LIN {X -0.105,Y -299.995,Z 1739.508,A 0.000,B 0.000,C 90.000,E1 271.547} C_DIS
LIN {X -0.094,Y -289.152,Z 1739.507,A 0.000,B 0.000,C 90.000,E1 271.260} C_DIS
LIN {X -0.103,Y -276.677,Z 1739.506,A 0.000,B 0.000,C 90.000,E1 271.031} C_DIS
LIN {X -0.110,Y -262.609,Z 1739.505,A 0.000,B 0.000,C 90.000,E1 270.859} C_DIS
LIN {X -0.020,Y -246.095,Z 1739.504,A 0.000,B 0.000,C 90.000,E1 270.688} C_DIS
LIN {X 0.079,Y -238.061,Z 1739.504,A 0.000,B 0.000,C 90.000,E1 270.630} C_DIS
LIN {X 0.025,Y -181.540,Z 1739.504,A 0.000,B 0.000,C 90.000,E1 270.630} C_DIS
LIN {X -0.061,Y -181.505,Z 1739.499,A 0.000,B 0.000,C 90.000,E1 269.771} C_DIS
LIN {X 0.044,Y -180.908,Z 1739.475,A 0.000,B 0.000,C 90.000,E1 265.527} C_DIS
LIN {X -0.079,Y -180.767,Z 1739.471,A 0.000,B 0.000,C 90.000,E1 264.723} C_DIS
LIN {X -0.008,Y -178.861,Z 1739.442,A 0.000,B 0.000,C 90.000,E1 259.634} C_DIS
LIN {X 0.064,Y -175.904,Z 1739.414,A 0.000,B 0.000,C 90.000,E1 254.519} C_DIS
LIN {X 0.003,Y -174.586,Z 1739.405,A 0.000,B 0.000,C 90.000,E1 252.834} C_DIS
LIN {X 0.037,Y -171.569,Z 1739.381,A 0.000,B 0.000,C 90.000,E1 248.539} C_DIS
LIN {X 0.019,Y -167.793,Z 1739.357,A 0.000,B 0.000,C 90.000,E1 244.229} C_DIS
LIN {X 0.033,Y -166.508,Z 1739.347,A 0.000,B 0.000,C 90.000,E1 242.487} C_DIS
LIN {X 0.029,Y -163.216,Z 1739.328,A 0.000,B 0.000,C 90.000,E1 238.997} C_DIS
LIN {X -0.006,Y -161.182,Z 1739.313,A 0.000,B 0.000,C 90.000,E1 236.373} C_DIS
LIN {X -0.006,Y -157.195,Z 1739.289,A 0.000,B 0.000,C 90.000,E1 231.949} C_DIS
LIN {X 0.040,Y -155.924,Z 1739.279,A 0.000,B 0.000,C 90.000,E1 230.150} C_DIS
LIN {X -0.011,Y -152.175,Z 1739.254,A 0.000,B 0.000,C 90.000,E1 225.688} C_DIS
LIN {X 0.005,Y -150.423,Z 1739.239,A 0.000,B 0.000,C 90.000,E1 222.975} C_DIS
LIN {X -0.070,Y -147.151,Z 1739.214,A 0.000,B 0.000,C 90.000,E1 218.463} C_DIS
LIN {X 0.018,Y -145.164,Z 1739.193,A 0.000,B 0.000,C 90.000,E1 214.771} C_DIS
LIN {X -0.066,Y -142.318,Z 1739.162,A 0.000,B 0.000,C 90.000,E1 209.283} C_DIS
LIN {X 0.054,Y -141.707,Z 1739.152,A 0.000,B 0.000,C 90.000,E1 207.385} C_DIS
LIN {X -0.023,Y -139.469,Z 1739.116,A 0.000,B 0.000,C 90.000,E1 200.918} C_DIS
LIN {X 0.031,Y -139.202,Z 1739.106,A 0.000,B 0.000,C 90.000,E1 199.033} C_DIS
LIN {X -0.042,Y -138.328,Z 1739.054,A 0.000,B 0.000,C 90.000,E1 189.726} C_DIS
LIN {X -0.039,Y -139.442,Z 1739.007,A 0.000,B 0.000,C 90.000,E1 181.318} C_DIS
LIN {X 0.040,Y -140.976,Z 1738.976,A 0.000,B 0.000,C 90.000,E1 175.698} C_DIS
LIN {X -0.010,Y -142.732,Z 1738.956,A 0.000,B 0.000,C 90.000,E1 172.008} C_DIS
LIN {X -0.053,Y -145.120,Z 1738.930,A 0.000,B 0.000,C 90.000,E1 167.409} C_DIS
LIN {X -0.058,Y -147.744,Z 1738.910,A 0.000,B 0.000,C 90.000,E1 163.740} C_DIS
LIN {X 0.023,Y -150.410,Z 1738.889,A 0.000,B 0.000,C 90.000,E1 160.061} C_DIS
LIN {X 0.038,Y -153.849,Z 1738.869,A 0.000,B 0.000,C 90.000,E1 156.433} C_DIS
LIN {X -0.044,Y -157.259,Z 1738.849,A 0.000,B 0.000,C 90.000,E1 152.871} C_DIS
LIN {X 0.034,Y -161.434,Z 1738.829,A 0.000,B 0.000,C 90.000,E1 149.282} C_DIS
LIN {X 0.041,Y -165.635,Z 1738.810,A 0.000,B 0.000,C 90.000,E1 145.754} C_DIS
LIN {X 0.024,Y -170.566,Z 1738.790,A 0.000,B 0.000,C 90.000,E1 142.271} C_DIS
LIN {X -0.069,Y -175.444,Z 1738.771,A 0.000,B 0.000,C 90.000,E1 138.852} C_DIS
LIN {X 0.047,Y -181.067,Z 1738.752,A 0.000,B 0.000,C 90.000,E1 135.405} C_DIS
LIN {X 0.038,Y -186.506,Z 1738.734,A 0.000,B 0.000,C 90.000,E1 132.043} C_DIS
LIN {X -0.020,Y -191.124,Z 1738.720,A 0.000,B 0.000,C 90.000,E1 129.564} C_DIS
LIN {X -0.099,Y -196.922,Z 1738.702,A 0.000,B 0.000,C 90.000,E1 126.297} C_DIS
LIN {X 0.095,Y -200.185,Z 1738.692,A 0.000,B 0.000,C 90.000,E1 124.612} C_DIS
LIN {X 0.091,Y -207.680,Z 1738.670,A 0.000,B 0.000,C 90.000,E1 120.590} C_DIS
LIN {X 0.056,Y -210.159,Z 1738.663,A 0.000,B 0.000,C 90.000,E1 119.411} C_DIS
LIN {X 0.030,Y -335.745,Z 1738.663,A 0.000,B 0.000,C 90.000,E1 119.411} C_DIS
LIN {X -0.088,Y -336.892,Z 1738.663,A 0.000,B 0.000,C 90.000,E1 119.411} C_DIS
LIN {X 0.032,Y -341.306,Z 1738.662,A 0.000,B 0.000,C 90.000,E1 119.205} C_DIS
LIN {X -0.012,Y -343.768,Z 1738.661,A 0.000,B 0.000,C 90.000,E1 119.027} C_DIS
LIN {X 0.124,Y -347.586,Z 1738.659,A 0.000,B 0.000,C 90.000,E1 118.565} C_DIS
LIN {X 0.008,Y -349.403,Z 1738.657,A 0.000,B 0.000,C 90.000,E1 118.281} C_DIS
LIN {X -0.092,Y -363.937,Z 1738.640,A 0.000,B 0.000,C 90.000,E1 115.283} C_DIS
LIN {X -0.172,Y -378.581,Z 1738.626,A 0.000,B 0.000,C 90.000,E1 112.642} C_DIS
LIN {X 0.064,Y -392.989,Z 1738.613,A 0.000,B 0.000,C 90.000,E1 110.301} C_DIS
LIN {X 0.021,Y -408.810,Z 1738.600,A 0.000,B 0.000,C 90.000,E1 108.055} C_DIS
LIN {X 0.119,Y -426.155,Z 1738.588,A 0.000,B 0.000,C 90.000,E1 105.843} C_DIS
LIN {X 0.012,Y -445.138,Z 1738.576,A 0.000,B 0.000,C 90.000,E1 103.716} C_DIS
LIN {X -0.048,Y -465.129,Z 1738.565,A 0.000,B 0.000,C 90.000,E1 101.715} C_DIS
LIN {X 0.245,Y -488.252,Z 1738.554,A 0.000,B 0.000,C 90.000,E1 99.613} C_DIS
LIN {X 0.198,Y -509.263,Z 1738.544,A 0.000,B 0.000,C 90.000,E1 97.936} C_DIS
LIN {X -0.014,Y -511.312,Z 1738.543,A 0.000,B 0.000,C 90.000,E1 97.757} C_DIS
LIN {X -0.101,Y -513.130,Z 1738.542,A 0.000,B 0.000,C 90.000,E1 97.530} C_DIS
LIN {X -0.123,Y -514.495,Z 1738.540,A 0.000,B 0.000,C 90.000,E1 97.296} C_DIS
LIN {X 0.246,Y -516.219,Z 1738.538,A 0.000,B 0.000,C 90.000,E1 96.777} C_DIS
LIN {X 0.109,Y -516.821,Z 1738.535,A 0.000,B 0.000,C 90.000,E1 96.315} C_DIS
LIN {X -0.018,Y -516.401,Z 1738.532,A 0.000,B 0.000,C 90.000,E1 95.853} C_DIS
LIN {X -0.144,Y -514.889,Z 1738.530,A 0.000,B 0.000,C 90.000,E1 95.391} C_DIS
LIN {X -0.231,Y -513.638,Z 1738.529,A 0.000,B 0.000,C 90.000,E1 95.163} C_DIS
LIN {X -0.048,Y -506.557,Z 1738.523,A 0.000,B 0.000,C 90.000,E1 94.188} C_DIS
LIN {X 0.214,Y -493.994,Z 1738.514,A 0.000,B 0.000,C 90.000,E1 92.465} C_DIS
LIN {X 0.190,Y -481.184,Z 1738.504,A 0.000,B 0.000,C 90.000,E1 90.745} C_DIS
LIN {X -0.083,Y -468.423,Z 1738.495,A 0.000,B 0.000,C 90.000,E1 89.026} C_DIS
LIN {X -0.131,Y -455.598,Z 1738.485,A 0.000,B 0.000,C 90.000,E1 87.249} C_DIS
LIN {X -0.184,Y -440.878,Z 1738.473,A 0.000,B 0.000,C 90.000,E1 85.179} C_DIS
LIN {X -0.140,Y -426.340,Z 1738.461,A 0.000,B 0.000,C 90.000,E1 83.053} C_DIS
LIN {X 0.132,Y -412.110,Z 1738.449,A 0.000,B 0.000,C 90.000,E1 80.849} C_DIS
LIN {X -0.002,Y -393.593,Z 1738.432,A 0.000,B 0.000,C 90.000,E1 77.813} C_DIS
LIN {X 0.145,Y -379.296,Z 1738.418,A 0.000,B 0.000,C 90.000,E1 75.227} C_DIS
LIN {X 0.106,Y -366.952,Z 1738.405,A 0.000,B 0.000,C 90.000,E1 72.906} C_DIS
LIN {X 0.045,Y -353.403,Z 1738.390,A 0.000,B 0.000,C 90.000,E1 70.242} C_DIS
LIN {X -0.120,Y -339.176,Z 1738.373,A 0.000,B 0.000,C 90.000,E1 67.230} C_DIS
LIN {X -0.058,Y -329.410,Z 1738.361,A 0.000,B 0.000,C 90.000,E1 65.049} C_DIS
LIN {X -0.200,Y -317.141,Z 1738.346,A 0.000,B 0.000,C 90.000,E1 62.231} C_DIS
LIN {X 0.050,Y -308.892,Z 1738.335,A 0.000,B 0.000,C 90.000,E1 60.255} C_DIS
LIN {X -0.098,Y -299.064,Z 1738.322,A 0.000,B 0.000,C 90.000,E1 57.995} C_DIS
LIN {X -0.130,Y -290.650,Z 1738.311,A 0.000,B 0.000,C 90.000,E1 56.008} C_DIS
LIN {X -0.073,Y -279.311,Z 1738.296,A 0.000,B 0.000,C 90.000,E1 53.290} C_DIS
LIN {X -0.108,Y -269.573,Z 1738.283,A 0.000,B 0.000,C 90.000,E1 50.884} C_DIS
LIN {X 0.030,Y -258.557,Z 1738.267,A 0.000,B 0.000,C 90.000,E1 48.038} C_DIS
LIN {X 0.032,Y -246.674,Z 1738.249,A 0.000,B 0.000,C 90.000,E1 44.798} C_DIS
LIN {X 0.070,Y -235.223,Z 1738.230,A 0.000,B 0.000,C 90.000,E1 41.472} C_DIS
LIN {X -0.002,Y -224.589,Z 1738.212,A 0.000,B 0.000,C 90.000,E1 38.096} C_DIS
LIN {X 0.061,Y -216.983,Z 1738.197,A 0.000,B 0.000,C 90.000,E1 35.391} C_DIS
LIN {X -0.014,Y -209.076,Z 1738.179,A 0.000,B 0.000,C 90.000,E1 32.291} C_DIS
LIN {X -0.045,Y -201.878,Z 1738.162,A 0.000,B 0.000,C 90.000,E1 29.127} C_DIS
LIN {X -0.026,Y -195.427,Z 1738.144,A 0.000,B 0.000,C 90.000,E1 25.899} C_DIS
LIN {X -0.061,Y -189.668,Z 1738.126,A 0.000,B 0.000,C 90.000,E1 22.642} C_DIS
LIN {X -0.030,Y -184.611,Z 1738.107,A 0.000,B 0.000,C 90.000,E1 19.322} C_DIS
LIN {X -0.010,Y -180.336,Z 1738.089,A 0.000,B 0.000,C 90.000,E1 15.969} C_DIS
LIN {X -0.016,Y -176.826,Z 1738.070,A 0.000,B 0.000,C 90.000,E1 12.591} C_DIS
LIN {X -0.049,Y -173.545,Z 1738.046,A 0.000,B 0.000,C 90.000,E1 8.341} C_DIS
LIN {X 0.048,Y -170.771,Z 1738.018,A 0.000,B 0.000,C 90.000,E1 3.154} C_DIS
LIN {X 0.062,Y -169.444,Z 1737.973,A 0.000,B 0.000,C 90.000,E1 355.184} C_DIS
LIN {X 0.057,Y -170.840,Z 1737.925,A 0.000,B 0.000,C 90.000,E1 346.533} C_DIS
LIN {X -0.063,Y -173.212,Z 1737.897,A 0.000,B 0.000,C 90.000,E1 341.402} C_DIS
LIN {X -0.019,Y -176.360,Z 1737.873,A 0.000,B 0.000,C 90.000,E1 337.102} C_DIS
LIN {X -0.085,Y -180.284,Z 1737.849,A 0.000,B 0.000,C 90.000,E1 332.871} C_DIS
LIN {X 0.040,Y -184.267,Z 1737.830,A 0.000,B 0.000,C 90.000,E1 329.459} C_DIS
LIN {X -0.017,Y -189.155,Z 1737.812,A 0.000,B 0.000,C 90.000,E1 326.135} C_DIS
LIN {X -0.060,Y -194.994,Z 1737.793,A 0.000,B 0.000,C 90.000,E1 322.844} C_DIS
LIN {X 0.072,Y -200.201,Z 1737.780,A 0.000,B 0.000,C 90.000,E1 320.356} C_DIS
LIN {X 0.032,Y -208.197,Z 1737.762,A 0.000,B 0.000,C 90.000,E1 317.148} C_DIS
LIN {X -0.005,Y -216.267,Z 1737.747,A 0.000,B 0.000,C 90.000,E1 314.393} C_DIS
LIN {X -0.010,Y -222.842,Z 1737.736,A 0.000,B 0.000,C 90.000,E1 312.447} C_DIS
LIN {X -0.110,Y -231.851,Z 1737.723,A 0.000,B 0.000,C 90.000,E1 310.172} C_DIS
LIN {X 0.024,Y -240.419,Z 1737.713,A 0.000,B 0.000,C 90.000,E1 308.257} C_DIS
LIN {X 0.160,Y -251.924,Z 1737.700,A 0.000,B 0.000,C 90.000,E1 306.011} C_DIS
LIN {X 0.122,Y -266.927,Z 1737.686,A 0.000,B 0.000,C 90.000,E1 303.499} C_DIS
LIN {X 0.083,Y -285.648,Z 1737.671,A 0.000,B 0.000,C 90.000,E1 300.718} C_DIS
LIN {X 0.081,Y -303.306,Z 1737.658,A 0.000,B 0.000,C 90.000,E1 298.359} C_DIS
LIN {X -0.094,Y -321.696,Z 1737.645,A 0.000,B 0.000,C 90.000,E1 296.104} C_DIS
LIN {X -0.079,Y -334.482,Z 1737.636,A 0.000,B 0.000,C 90.000,E1 294.567} C_DIS
LIN {X -0.023,Y -347.643,Z 1737.628,A 0.000,B 0.000,C 90.000,E1 293.003} C_DIS
LIN {X 0.095,Y -357.760,Z 1737.621,A 0.000,B 0.000,C 90.000,E1 291.770} C_DIS
LIN {X -0.150,Y -367.553,Z 1737.614,A 0.000,B 0.000,C 90.000,E1 290.610} C_DIS
LIN {X -0.022,Y -374.523,Z 1737.609,A 0.000,B 0.000,C 90.000,E1 289.704} C_DIS
LIN {X 0.183,Y -378.791,Z 1737.606,A 0.000,B 0.000,C 90.000,E1 289.087} C_DIS
LIN {X -0.066,Y -382.655,Z 1737.603,A 0.000,B 0.000,C 90.000,E1 288.544} C_DIS
LIN {X 0.071,Y -386.084,Z 1737.600,A 0.000,B 0.000,C 90.000,E1 287.946} C_DIS
LIN {X -0.136,Y -389.068,Z 1737.597,A 0.000,B 0.000,C 90.000,E1 287.402} C_DIS
LIN {X 0.047,Y -391.609,Z 1737.593,A 0.000,B 0.000,C 90.000,E1 286.804} C_DIS
LIN {X -0.078,Y -394.658,Z 1737.589,A 0.000,B 0.000,C 90.000,E1 285.969} C_DIS
LIN {X 0.139,Y -396.227,Z 1737.585,A 0.000,B 0.000,C 90.000,E1 285.371} C_DIS
LIN {X -0.017,Y -397.450,Z 1737.582,A 0.000,B 0.000,C 90.000,E1 284.828} C_DIS
LIN {X 0.118,Y -398.340,Z 1737.579,A 0.000,B 0.000,C 90.000,E1 284.245} C_DIS
LIN {X -0.027,Y -398.898,Z 1737.576,A 0.000,B 0.000,C 90.000,E1 283.703} C_DIS
LIN {X 0.125,Y -399.041,Z 1737.573,A 0.000,B 0.000,C 90.000,E1 283.119} C_DIS
LIN {X -0.107,Y -398.829,Z 1737.570,A 0.000,B 0.000,C 90.000,E1 282.591} C_DIS
LIN {X 0.052,Y -398.155,Z 1737.567,A 0.000,B 0.000,C 90.000,E1 282.007} C_DIS
LIN {X -0.178,Y -397.045,Z 1737.564,A 0.000,B 0.000,C 90.000,E1 281.478} C_DIS
LIN {X -0.025,Y -395.355,Z 1737.561,A 0.000,B 0.000,C 90.000,E1 280.894} C_DIS
LIN {X 0.120,Y -393.108,Z 1737.557,A 0.000,B 0.000,C 90.000,E1 280.310} C_DIS
LIN {X -0.139,Y -390.215,Z 1737.554,A 0.000,B 0.000,C 90.000,E1 279.782} C_DIS
LIN {X -0.026,Y -381.971,Z 1737.546,A 0.000,B 0.000,C 90.000,E1 278.341} C_DIS
LIN {X 0.051,Y -377.336,Z 1737.542,A 0.000,B 0.000,C 90.000,E1 277.466} C_DIS
LIN {X 0.027,Y -373.748,Z 1737.538,A 0.000,B 0.000,C 90.000,E1 276.891} C_DIS
LIN {X -0.017,Y -369.584,Z 1737.535,A 0.000,B 0.000,C 90.000,E1 276.315} C_DIS
LIN {X -0.080,Y -364.671,Z 1737.532,A 0.000,B 0.000,C 90.000,E1 275.739} C_DIS
LIN {X -0.168,Y -358.972,Z 1737.529,A 0.000,B 0.000,C 90.000,E1 275.163} C_DIS
LIN {X 0.052,Y -353.211,Z 1737.526,A 0.000,B 0.000,C 90.000,E1 274.588} C_DIS
LIN {X 0.112,Y -344.344,Z 1737.521,A 0.000,B 0.000,C 90.000,E1 273.841} C_DIS
LIN {X 0.146,Y -338.207,Z 1737.519,A 0.000,B 0.000,C 90.000,E1 273.383} C_DIS
LIN {X 0.047,Y -331.920,Z 1737.517,A 0.000,B 0.000,C 90.000,E1 272.980} C_DIS
LIN {X 0.117,Y -325.356,Z 1737.514,A 0.000,B 0.000,C 90.000,E1 272.579} C_DIS
LIN {X 0.077,Y -318.598,Z 1737.512,A 0.000,B 0.000,C 90.000,E1 272.236} C_DIS
LIN {X -0.028,Y -311.635,Z 1737.511,A 0.000,B 0.000,C 90.000,E1 271.949} C_DIS
LIN {X 0.119,Y -304.471,Z 1737.509,A 0.000,B 0.000,C 90.000,E1 271.661} C_DIS
LIN {X -0.056,Y -293.557,Z 1737.508,A 0.000,B 0.000,C 90.000,E1 271.375} C_DIS
LIN {X -0.060,Y -286.006,Z 1737.507,A 0.000,B 0.000,C 90.000,E1 271.203} C_DIS
LIN {X 0.065,Y -273.757,Z 1737.505,A 0.000,B 0.000,C 90.000,E1 270.974} C_DIS
LIN {X 0.066,Y -259.464,Z 1737.505,A 0.000,B 0.000,C 90.000,E1 270.802} C_DIS
LIN {X 0.016,Y -243.753,Z 1737.504,A 0.000,B 0.000,C 90.000,E1 270.688} C_DIS
LIN {X -0.077,Y -236.046,Z 1737.504,A 0.000,B 0.000,C 90.000,E1 270.688} C_DIS
LIN {X 0.087,Y -181.536,Z 1737.504,A 0.000,B 0.000,C 90.000,E1 270.630} C_DIS
LIN {X 0.037,Y -181.513,Z 1737.499,A 0.000,B 0.000,C 90.000,E1 269.771} C_DIS
LIN {X -0.039,Y -180.908,Z 1737.475,A 0.000,B 0.000,C 90.000,E1 265.584} C_DIS
LIN {X 0.019,Y -180.779,Z 1737.471,A 0.000,B 0.000,C 90.000,E1 264.723} C_DIS
LIN {X -0.087,Y -178.875,Z 1737.443,A 0.000,B 0.000,C 90.000,E1 259.690} C_DIS
LIN {X -0.010,Y -175.918,Z 1737.414,A 0.000,B 0.000,C 90.000,E1 254.574} C_DIS
LIN {X 0.046,Y -174.613,Z 1737.405,A 0.000,B 0.000,C 90.000,E1 252.851} C_DIS
LIN {X -0.028,Y -171.593,Z 1737.381,A 0.000,B 0.000,C 90.000,E1 248.592} C_DIS
LIN {X -0.039,Y -167.815,Z 1737.357,A 0.000,B 0.000,C 90.000,E1 244.280} C_DIS
LIN {X -0.021,Y -166.538,Z 1737.347,A 0.000,B 0.000,C 90.000,E1 242.538} C_DIS
LIN {X 0.028,Y -162.536,Z 1737.323,A 0.000,B 0.000,C 90.000,E1 238.152} C_DIS
LIN {X -0.050,Y -161.212,Z 1737.313,A 0.000,B 0.000,C 90.000,E1 236.421} C_DIS
LIN {X -0.014,Y -157.220,Z 1737.289,A 0.000,B 0.000,C 90.000,E1 231.984} C_DIS
LIN {X 0.009,Y -155.946,Z 1737.279,A 0.000,B 0.000,C 90.000,E1 230.194} C_DIS
LIN {X -0.032,Y -152.199,Z 1737.254,A 0.000,B 0.000,C 90.000,E1 225.729} C_DIS
LIN {X -0.010,Y -150.444,Z 1737.239,A 0.000,B 0.000,C 90.000,E1 223.014} C_DIS
LIN {X 0.016,Y -147.171,Z 1737.214,A 0.000,B 0.000,C 90.000,E1 218.463} C_DIS
LIN {X -0.016,Y -145.187,Z 1737.193,A 0.000,B 0.000,C 90.000,E1 214.818} C_DIS
LIN {X 0.018,Y -142.331,Z 1737.163,A 0.000,B 0.000,C 90.000,E1 209.283} C_DIS
LIN {X -0.053,Y -141.719,Z 1737.152,A 0.000,B 0.000,C 90.000,E1 207.462} C_DIS
LIN {X 0.060,Y -139.476,Z 1737.116,A 0.000,B 0.000,C 90.000,E1 200.918} C_DIS
LIN {X 0.051,Y -138.973,Z 1737.101,A 0.000,B 0.000,C 90.000,E1 198.127} C_DIS
LIN {X 0.040,Y -138.331,Z 1737.054,A 0.000,B 0.000,C 90.000,E1 189.726} C_DIS
LIN {X 0.044,Y -139.434,Z 1737.007,A 0.000,B 0.000,C 90.000,E1 181.318} C_DIS
LIN {X -0.016,Y -140.963,Z 1736.976,A 0.000,B 0.000,C 90.000,E1 175.755} C_DIS
LIN {X 0.074,Y -142.719,Z 1736.956,A 0.000,B 0.000,C 90.000,E1 172.008} C_DIS
LIN {X 0.033,Y -145.098,Z 1736.930,A 0.000,B 0.000,C 90.000,E1 167.409} C_DIS
LIN {X 0.029,Y -147.723,Z 1736.910,A 0.000,B 0.000,C 90.000,E1 163.740} C_DIS
LIN {X -0.032,Y -150.382,Z 1736.889,A 0.000,B 0.000,C 90.000,E1 160.115} C_DIS
LIN {X -0.013,Y -153.813,Z 1736.869,A 0.000,B 0.000,C 90.000,E1 156.485} C_DIS
LIN {X 0.046,Y -157.224,Z 1736.849,A 0.000,B 0.000,C 90.000,E1 152.871} C_DIS
LIN {X -0.014,Y -161.392,Z 1736.830,A 0.000,B 0.000,C 90.000,E1 149.331} C_DIS
LIN {X -0.003,Y -165.594,Z 1736.810,A 0.000,B 0.000,C 90.000,E1 145.801} C_DIS
LIN {X -0.017,Y -170.517,Z 1736.791,A 0.000,B 0.000,C 90.000,E1 142.316} C_DIS
LIN {X 0.027,Y -175.396,Z 1736.771,A 0.000,B 0.000,C 90.000,E1 138.852} C_DIS
LIN {X 0.018,Y -181.021,Z 1736.753,A 0.000,B 0.000,C 90.000,E1 135.445} C_DIS
LIN {X 0.012,Y -186.452,Z 1736.734,A 0.000,B 0.000,C 90.000,E1 132.081} C_DIS
LIN {X 0.081,Y -191.076,Z 1736.720,A 0.000,B 0.000,C 90.000,E1 129.564} C_DIS
LIN {X 0.004,Y -196.865,Z 1736.702,A 0.000,B 0.000,C 90.000,E1 126.297} C_DIS
LIN {X -0.080,Y -200.123,Z 1736.693,A 0.000,B 0.000,C 90.000,E1 124.692} C_DIS
LIN {X -0.087,Y -207.620,Z 1736.670,A 0.000,B 0.000,C 90.000,E1 120.669} C_DIS
LIN {X -0.021,Y -210.103,Z 1736.664,A 0.000,B 0.000,C 90.000,E1 119.461} C_DIS
LIN {X -0.093,Y -335.517,Z 1736.664,A 0.000,B 0.000,C 90.000,E1 119.461} C_DIS
LIN {X 0.081,Y -336.703,Z 1736.663,A 0.000,B 0.000,C 90.000,E1 119.411} C_DIS
LIN {X 0.205,Y -341.146,Z 1736.662,A 0.000,B 0.000,C 90.000,E1 119.205} C_DIS
LIN {X -0.139,Y -343.611,Z 1736.661,A 0.000,B 0.000,C 90.000,E1 119.077} C_DIS
LIN {X -0.001,Y -347.427,Z 1736.659,A 0.000,B 0.000,C 90.000,E1 118.615} C_DIS
LIN {X 0.024,Y -349.245,Z 1736.657,A 0.000,B 0.000,C 90.000,E1 118.309} C_DIS
LIN {X 0.093,Y -363.763,Z 1736.641,A 0.000,B 0.000,C 90.000,E1 115.283} C_DIS
LIN {X 0.015,Y -378.390,Z 1736.626,A 0.000,B 0.000,C 90.000,E1 112.642} C_DIS
LIN {X -0.114,Y -392.781,Z 1736.613,A 0.000,B 0.000,C 90.000,E1 110.355} C_DIS
LIN {X 0.213,Y -408.585,Z 1736.600,A 0.000,B 0.000,C 90.000,E1 108.055} C_DIS
LIN {X -0.096,Y -425.910,Z 1736.588,A 0.000,B 0.000,C 90.000,E1 105.898} C_DIS
LIN {X -0.226,Y -444.875,Z 1736.576,A 0.000,B 0.000,C 90.000,E1 103.772} C_DIS
LIN {X 0.138,Y -464.859,Z 1736.565,A 0.000,B 0.000,C 90.000,E1 101.715} C_DIS
LIN {X -0.060,Y -487.976,Z 1736.554,A 0.000,B 0.000,C 90.000,E1 99.670} C_DIS
LIN {X -0.137,Y -508.985,Z 1736.544,A 0.000,B 0.000,C 90.000,E1 97.992} C_DIS
LIN {X 0.154,Y -511.042,Z 1736.543,A 0.000,B 0.000,C 90.000,E1 97.757} C_DIS
LIN {X 0.069,Y -512.860,Z 1736.542,A 0.000,B 0.000,C 90.000,E1 97.530} C_DIS
LIN {X 0.052,Y -514.227,Z 1736.541,A 0.000,B 0.000,C 90.000,E1 97.296} C_DIS
LIN {X -0.093,Y -515.957,Z 1736.538,A 0.000,B 0.000,C 90.000,E1 96.834} C_DIS
LIN {X -0.231,Y -516.566,Z 1736.535,A 0.000,B 0.000,C 90.000,E1 96.372} C_DIS
LIN {X 0.152,Y -516.154,Z 1736.533,A 0.000,B 0.000,C 90.000,E1 95.853} C_DIS
LIN {X 0.025,Y -514.651,Z 1736.530,A 0.000,B 0.000,C 90.000,E1 95.391} C_DIS
LIN {X -0.063,Y -513.406,Z 1736.529,A 0.000,B 0.000,C 90.000,E1 95.163} C_DIS
LIN {X 0.114,Y -506.330,Z 1736.523,A 0.000,B 0.000,C 90.000,E1 94.188} C_DIS
LIN {X -0.126,Y -493.770,Z 1736.514,A 0.000,B 0.000,C 90.000,E1 92.522} C_DIS
LIN {X -0.145,Y -480.954,Z 1736.504,A 0.000,B 0.000,C 90.000,E1 90.802} C_DIS
LIN {X 0.055,Y -468.194,Z 1736.495,A 0.000,B 0.000,C 90.000,E1 89.026} C_DIS
LIN {X -0.001,Y -455.379,Z 1736.485,A 0.000,B 0.000,C 90.000,E1 87.249} C_DIS
LIN {X 0.162,Y -442.465,Z 1736.475,A 0.000,B 0.000,C 90.000,E1 85.412} C_DIS
LIN {X 0.092,Y -429.699,Z 1736.464,A 0.000,B 0.000,C 90.000,E1 83.571} C_DIS
LIN {X -0.177,Y -417.136,Z 1736.454,A 0.000,B 0.000,C 90.000,E1 81.724} C_DIS
LIN {X 0.155,Y -398.215,Z 1736.437,A 0.000,B 0.000,C 90.000,E1 78.645} C_DIS
LIN {X 0.039,Y -383.704,Z 1736.423,A 0.000,B 0.000,C 90.000,E1 76.117} C_DIS
LIN {X 0.108,Y -371.237,Z 1736.410,A 0.000,B 0.000,C 90.000,E1 73.795} C_DIS
LIN {X -0.011,Y -359.030,Z 1736.397,A 0.000,B 0.000,C 90.000,E1 71.456} C_DIS
LIN {X -0.132,Y -344.398,Z 1736.380,A 0.000,B 0.000,C 90.000,E1 68.465} C_DIS
LIN {X -0.086,Y -334.637,Z 1736.368,A 0.000,B 0.000,C 90.000,E1 66.305} C_DIS
LIN {X 0.060,Y -322.128,Z 1736.353,A 0.000,B 0.000,C 90.000,E1 63.461} C_DIS
LIN {X -0.030,Y -313.999,Z 1736.342,A 0.000,B 0.000,C 90.000,E1 61.563} C_DIS
LIN {X 0.045,Y -304.268,Z 1736.329,A 0.000,B 0.000,C 90.000,E1 59.282} C_DIS
LIN {X -0.048,Y -294.502,Z 1736.317,A 0.000,B 0.000,C 90.000,E1 56.993} C_DIS
LIN {X -0.009,Y -286.033,Z 1736.305,A 0.000,B 0.000,C 90.000,E1 54.975} C_DIS
LIN {X -0.130,Y -274.840,Z 1736.290,A 0.000,B 0.000,C 90.000,E1 52.271} C_DIS
LIN {X -0.094,Y -265.096,Z 1736.277,A 0.000,B 0.000,C 90.000,E1 49.828} C_DIS
LIN {X -0.084,Y -254.181,Z 1736.261,A 0.000,B 0.000,C 90.000,E1 46.986} C_DIS
LIN {X 0.166,Y -243.715,Z 1736.245,A 0.000,B 0.000,C 90.000,E1 44.028} C_DIS
LIN {X -0.054,Y -232.449,Z 1736.226,A 0.000,B 0.000,C 90.000,E1 40.744} C_DIS
LIN {X 0.006,Y -222.009,Z 1736.207,A 0.000,B 0.000,C 90.000,E1 37.317} C_DIS
LIN {X 0.022,Y -214.644,Z 1736.192,A 0.000,B 0.000,C 90.000,E1 34.612} C_DIS
LIN {X 0.062,Y -206.948,Z 1736.175,A 0.000,B 0.000,C 90.000,E1 31.465} C_DIS
LIN {X 0.047,Y -199.982,Z 1736.157,A 0.000,B 0.000,C 90.000,E1 28.281} C_DIS
LIN {X -0.068,Y -193.740,Z 1736.139,A 0.000,B 0.000,C 90.000,E1 25.079} C_DIS
LIN {X 0.030,Y -188.141,Z 1736.121,A 0.000,B 0.000,C 90.000,E1 21.770} C_DIS
LIN {X -0.045,Y -183.331,Z 1736.103,A 0.000,B 0.000,C 90.000,E1 18.471} C_DIS
LIN {X -0.108,Y -179.237,Z 1736.084,A 0.000,B 0.000,C 90.000,E1 15.134} C_DIS
LIN {X -0.008,Y -175.952,Z 1736.065,A 0.000,B 0.000,C 90.000,E1 11.715} C_DIS
LIN {X -0.072,Y -172.842,Z 1736.041,A 0.000,B 0.000,C 90.000,E1 7.466} C_DIS
LIN {X -0.038,Y -170.324,Z 1736.013,A 0.000,B 0.000,C 90.000,E1 2.293} C_DIS
LIN {X 0.057,Y -169.274,Z 1735.969,A 0.000,B 0.000,C 90.000,E1 354.318} C_DIS
LIN {X -0.049,Y -170.993,Z 1735.920,A 0.000,B 0.000,C 90.000,E1 345.700} C_DIS
LIN {X 0.055,Y -173.609,Z 1735.892,A 0.000,B 0.000,C 90.000,E1 340.496} C_DIS
LIN {X 0.015,Y -176.980,Z 1735.868,A 0.000,B 0.000,C 90.000,E1 336.230} C_DIS
LIN {X 0.045,Y -181.115,Z 1735.844,A 0.000,B 0.000,C 90.000,E1 331.975} C_DIS
LIN {X 0.029,Y -185.352,Z 1735.826,A 0.000,B 0.000,C 90.000,E1 328.614} C_DIS
LIN {X -0.061,Y -190.485,Z 1735.807,A 0.000,B 0.000,C 90.000,E1 325.308} C_DIS
LIN {X -0.095,Y -195.037,Z 1735.793,A 0.000,B 0.000,C 90.000,E1 322.844} C_DIS
LIN {X 0.052,Y -202.180,Z 1735.775,A 0.000,B 0.000,C 90.000,E1 319.542} C_DIS
LIN {X 0.032,Y -209.428,Z 1735.760,A 0.000,B 0.000,C 90.000,E1 316.743} C_DIS
LIN {X 0.124,Y -216.432,Z 1735.747,A 0.000,B 0.000,C 90.000,E1 314.352} C_DIS
LIN {X -0.034,Y -223.033,Z 1735.736,A 0.000,B 0.000,C 90.000,E1 312.447} C_DIS
LIN {X -0.074,Y -230.467,Z 1735.725,A 0.000,B 0.000,C 90.000,E1 310.539} C_DIS
LIN {X 0.032,Y -238.788,Z 1735.715,A 0.000,B 0.000,C 90.000,E1 308.624} C_DIS
LIN {X -0.066,Y -250.065,Z 1735.702,A 0.000,B 0.000,C 90.000,E1 306.423} C_DIS
LIN {X -0.079,Y -260.471,Z 1735.692,A 0.000,B 0.000,C 90.000,E1 304.612} C_DIS
LIN {X 0.088,Y -278.636,Z 1735.677,A 0.000,B 0.000,C 90.000,E1 301.750} C_DIS
LIN {X 0.068,Y -298.424,Z 1735.661,A 0.000,B 0.000,C 90.000,E1 299.027} C_DIS
LIN {X -0.009,Y -319.260,Z 1735.647,A 0.000,B 0.000,C 90.000,E1 296.411} C_DIS
LIN {X -0.149,Y -331.997,Z 1735.638,A 0.000,B 0.000,C 90.000,E1 294.899} C_DIS
LIN {X -0.110,Y -345.202,Z 1735.630,A 0.000,B 0.000,C 90.000,E1 293.334} C_DIS
LIN {X 0.090,Y -355.417,Z 1735.623,A 0.000,B 0.000,C 90.000,E1 292.078} C_DIS
LIN {X -0.121,Y -367.725,Z 1735.614,A 0.000,B 0.000,C 90.000,E1 290.610} C_DIS
LIN {X 0.009,Y -374.708,Z 1735.609,A 0.000,B 0.000,C 90.000,E1 289.704} C_DIS
LIN {X -0.141,Y -378.989,Z 1735.606,A 0.000,B 0.000,C 90.000,E1 289.141} C_DIS
LIN {X 0.091,Y -384.629,Z 1735.601,A 0.000,B 0.000,C 90.000,E1 288.236} C_DIS
LIN {X -0.126,Y -387.809,Z 1735.598,A 0.000,B 0.000,C 90.000,E1 287.692} C_DIS
LIN {X 0.046,Y -390.589,Z 1735.595,A 0.000,B 0.000,C 90.000,E1 287.094} C_DIS
LIN {X -0.137,Y -392.943,Z 1735.592,A 0.000,B 0.000,C 90.000,E1 286.551} C_DIS
LIN {X -0.038,Y -394.879,Z 1735.589,A 0.000,B 0.000,C 90.000,E1 285.969} C_DIS
LIN {X -0.201,Y -396.449,Z 1735.586,A 0.000,B 0.000,C 90.000,E1 285.426} C_DIS
LIN {X 0.026,Y -397.685,Z 1735.582,A 0.000,B 0.000,C 90.000,E1 284.828} C_DIS
LIN {X 0.164,Y -398.578,Z 1735.579,A 0.000,B 0.000,C 90.000,E1 284.245} C_DIS
LIN {X 0.020,Y -399.122,Z 1735.576,A 0.000,B 0.000,C 90.000,E1 283.703} C_DIS
LIN {X 0.173,Y -399.270,Z 1735.573,A 0.000,B 0.000,C 90.000,E1 283.119} C_DIS
LIN {X -0.057,Y -399.089,Z 1735.570,A 0.000,B 0.000,C 90.000,E1 282.591} C_DIS
LIN {X 0.103,Y -398.421,Z 1735.567,A 0.000,B 0.000,C 90.000,E1 282.007} C_DIS
LIN {X -0.127,Y -397.299,Z 1735.564,A 0.000,B 0.000,C 90.000,E1 281.478} C_DIS
LIN {X 0.028,Y -395.595,Z 1735.561,A 0.000,B 0.000,C 90.000,E1 280.894} C_DIS
LIN {X 0.175,Y -393.392,Z 1735.557,A 0.000,B 0.000,C 90.000,E1 280.310} C_DIS
LIN {X -0.149,Y -390.578,Z 1735.554,A 0.000,B 0.000,C 90.000,E1 279.792} C_DIS
LIN {X 0.055,Y -382.308,Z 1735.546,A 0.000,B 0.000,C 90.000,E1 278.341} C_DIS
LIN {X 0.108,Y -377.600,Z 1735.542,A 0.000,B 0.000,C 90.000,E1 277.473} C_DIS
LIN {X 0.132,Y -373.983,Z 1735.538,A 0.000,B 0.000,C 90.000,E1 276.891} C_DIS
LIN {X 0.090,Y -369.788,Z 1735.535,A 0.000,B 0.000,C 90.000,E1 276.315} C_DIS
LIN {X 0.026,Y -364.885,Z 1735.532,A 0.000,B 0.000,C 90.000,E1 275.739} C_DIS
LIN {X -0.063,Y -359.207,Z 1735.529,A 0.000,B 0.000,C 90.000,E1 275.163} C_DIS
LIN {X 0.002,Y -350.518,Z 1735.524,A 0.000,B 0.000,C 90.000,E1 274.359} C_DIS
LIN {X -0.070,Y -344.678,Z 1735.522,A 0.000,B 0.000,C 90.000,E1 273.898} C_DIS
LIN {X 0.130,Y -335.598,Z 1735.518,A 0.000,B 0.000,C 90.000,E1 273.212} C_DIS
LIN {X 0.090,Y -329.117,Z 1735.516,A 0.000,B 0.000,C 90.000,E1 272.808} C_DIS
LIN {X -0.064,Y -322.435,Z 1735.514,A 0.000,B 0.000,C 90.000,E1 272.465} C_DIS
LIN {X 0.013,Y -315.507,Z 1735.512,A 0.000,B 0.000,C 90.000,E1 272.121} C_DIS
LIN {X 0.033,Y -308.539,Z 1735.510,A 0.000,B 0.000,C 90.000,E1 271.835} C_DIS
LIN {X 0.033,Y -297.863,Z 1735.508,A 0.000,B 0.000,C 90.000,E1 271.489} C_DIS
LIN {X -0.054,Y -290.662,Z 1735.507,A 0.000,B 0.000,C 90.000,E1 271.318} C_DIS
LIN {X -0.051,Y -278.551,Z 1735.506,A 0.000,B 0.000,C 90.000,E1 271.088} C_DIS
LIN {X -0.088,Y -265.066,Z 1735.505,A 0.000,B 0.000,C 90.000,E1 270.917} C_DIS
LIN {X -0.045,Y -255.020,Z 1735.504,A 0.000,B 0.000,C 90.000,E1 270.802} C_DIS
LIN {X 0.046,Y -239.872,Z 1735.504,A 0.000,B 0.000,C 90.000,E1 270.688} C_DIS
LIN {X 0.001,Y -181.529,Z 1735.504,A 0.000,B 0.000,C 90.000,E1 270.688} C_DIS
LIN {X -0.046,Y -181.522,Z 1735.499,A 0.000,B 0.000,C 90.000,E1 269.828} C_DIS
LIN {X -0.063,Y -180.791,Z 1735.471,A 0.000,B 0.000,C 90.000,E1 264.780} C_DIS
LIN {X 0.011,Y -178.888,Z 1735.443,A 0.000,B 0.000,C 90.000,E1 259.690} C_DIS
LIN {X 0.087,Y -175.932,Z 1735.414,A 0.000,B 0.000,C 90.000,E1 254.574} C_DIS
LIN {X 0.033,Y -175.377,Z 1735.410,A 0.000,B 0.000,C 90.000,E1 253.740} C_DIS
LIN {X 0.030,Y -172.151,Z 1735.386,A 0.000,B 0.000,C 90.000,E1 249.464} C_DIS
LIN {X 0.067,Y -171.617,Z 1735.381,A 0.000,B 0.000,C 90.000,E1 248.592} C_DIS
LIN {X 0.055,Y -167.840,Z 1735.357,A 0.000,B 0.000,C 90.000,E1 244.280} C_DIS
LIN {X -0.004,Y -166.568,Z 1735.348,A 0.000,B 0.000,C 90.000,E1 242.564} C_DIS
LIN {X -0.018,Y -162.561,Z 1735.323,A 0.000,B 0.000,C 90.000,E1 238.201} C_DIS
LIN {X 0.042,Y -161.241,Z 1735.313,A 0.000,B 0.000,C 90.000,E1 236.421} C_DIS
LIN {X -0.047,Y -157.245,Z 1735.289,A 0.000,B 0.000,C 90.000,E1 232.029} C_DIS
LIN {X -0.001,Y -155.968,Z 1735.279,A 0.000,B 0.000,C 90.000,E1 230.231} C_DIS
LIN {X 0.057,Y -152.223,Z 1735.254,A 0.000,B 0.000,C 90.000,E1 225.729} C_DIS
LIN {X -0.032,Y -150.466,Z 1735.239,A 0.000,B 0.000,C 90.000,E1 223.056} C_DIS
LIN {X -0.012,Y -147.191,Z 1735.214,A 0.000,B 0.000,C 90.000,E1 218.508} C_DIS
LIN {X 0.069,Y -145.210,Z 1735.194,A 0.000,B 0.000,C 90.000,E1 214.818} C_DIS
LIN {X -0.021,Y -142.343,Z 1735.163,A 0.000,B 0.000,C 90.000,E1 209.333} C_DIS
LIN {X 0.032,Y -141.731,Z 1735.153,A 0.000,B 0.000,C 90.000,E1 207.462} C_DIS
LIN {X 0.014,Y -139.483,Z 1735.117,A 0.000,B 0.000,C 90.000,E1 200.972} C_DIS
LIN {X 0.003,Y -138.983,Z 1735.101,A 0.000,B 0.000,C 90.000,E1 198.181} C_DIS
LIN {X -0.035,Y -138.333,Z 1735.054,A 0.000,B 0.000,C 90.000,E1 189.792} C_DIS
LIN {X -0.012,Y -139.426,Z 1735.008,A 0.000,B 0.000,C 90.000,E1 181.375} C_DIS
LIN {X 0.042,Y -141.351,Z 1734.971,A 0.000,B 0.000,C 90.000,E1 174.837} C_DIS
LIN {X 0.019,Y -142.705,Z 1734.956,A 0.000,B 0.000,C 90.000,E1 172.064} C_DIS
LIN {X -0.023,Y -145.077,Z 1734.930,A 0.000,B 0.000,C 90.000,E1 167.465} C_DIS
LIN {X -0.027,Y -147.702,Z 1734.910,A 0.000,B 0.000,C 90.000,E1 163.795} C_DIS
LIN {X 0.006,Y -150.354,Z 1734.890,A 0.000,B 0.000,C 90.000,E1 160.134} C_DIS
LIN {X 0.076,Y -153.778,Z 1734.870,A 0.000,B 0.000,C 90.000,E1 156.485} C_DIS
LIN {X -0.003,Y -157.190,Z 1734.850,A 0.000,B 0.000,C 90.000,E1 152.922} C_DIS
LIN {X 0.078,Y -161.349,Z 1734.830,A 0.000,B 0.000,C 90.000,E1 149.331} C_DIS
LIN {X 0.090,Y -165.552,Z 1734.810,A 0.000,B 0.000,C 90.000,E1 145.801} C_DIS
LIN {X -0.025,Y -170.467,Z 1734.791,A 0.000,B 0.000,C 90.000,E1 142.351} C_DIS
LIN {X -0.008,Y -175.348,Z 1734.772,A 0.000,B 0.000,C 90.000,E1 138.895} C_DIS
LIN {X -0.012,Y -180.973,Z 1734.753,A 0.000,B 0.000,C 90.000,E1 135.486} C_DIS
LIN {X -0.024,Y -186.397,Z 1734.734,A 0.000,B 0.000,C 90.000,E1 132.123} C_DIS
LIN {X -0.085,Y -191.025,Z 1734.720,A 0.000,B 0.000,C 90.000,E1 129.644} C_DIS
LIN {X 0.107,Y -196.807,Z 1734.702,A 0.000,B 0.000,C 90.000,E1 126.297} C_DIS
LIN {X 0.026,Y -200.060,Z 1734.693,A 0.000,B 0.000,C 90.000,E1 124.692} C_DIS
LIN {X 0.020,Y -207.560,Z 1734.670,A 0.000,B 0.000,C 90.000,E1 120.669} C_DIS
LIN {X -0.017,Y -210.045,Z 1734.664,A 0.000,B 0.000,C 90.000,E1 119.489} C_DIS
LIN {X 0.078,Y -335.262,Z 1734.664,A 0.000,B 0.000,C 90.000,E1 119.461} C_DIS
LIN {X -0.040,Y -336.493,Z 1734.664,A 0.000,B 0.000,C 90.000,E1 119.461} C_DIS
LIN {X -0.085,Y -340.971,Z 1734.663,A 0.000,B 0.000,C 90.000,E1 119.283} C_DIS
LIN {X 0.038,Y -343.444,Z 1734.662,A 0.000,B 0.000,C 90.000,E1 119.077} C_DIS
LIN {X 0.186,Y -347.259,Z 1734.659,A 0.000,B 0.000,C 90.000,E1 118.615} C_DIS
LIN {X -0.093,Y -349.079,Z 1734.657,A 0.000,B 0.000,C 90.000,E1 118.359} C_DIS
LIN {X 0.023,Y -365.127,Z 1734.639,A 0.000,B 0.000,C 90.000,E1 115.027} C_DIS
LIN {X -0.017,Y -379.909,Z 1734.624,A 0.000,B 0.000,C 90.000,E1 112.386} C_DIS
LIN {X 0.117,Y -394.452,Z 1734.612,A 0.000,B 0.000,C 90.000,E1 110.066} C_DIS
LIN {X 0.119,Y -410.420,Z 1734.599,A 0.000,B 0.000,C 90.000,E1 107.819} C_DIS
LIN {X -0.146,Y -427.922,Z 1734.587,A 0.000,B 0.000,C 90.000,E1 105.662} C_DIS
LIN {X -0.199,Y -447.045,Z 1734.575,A 0.000,B 0.000,C 90.000,E1 103.536} C_DIS
LIN {X -0.139,Y -467.094,Z 1734.564,A 0.000,B 0.000,C 90.000,E1 101.535} C_DIS
LIN {X 0.187,Y -490.299,Z 1734.553,A 0.000,B 0.000,C 90.000,E1 99.443} C_DIS
LIN {X 0.047,Y -508.690,Z 1734.544,A 0.000,B 0.000,C 90.000,E1 97.992} C_DIS
LIN {X -0.169,Y -510.762,Z 1734.543,A 0.000,B 0.000,C 90.000,E1 97.814} C_DIS
LIN {X -0.248,Y -512.585,Z 1734.542,A 0.000,B 0.000,C 90.000,E1 97.587} C_DIS
LIN {X 0.250,Y -513.955,Z 1734.541,A 0.000,B 0.000,C 90.000,E1 97.296} C_DIS
LIN {X 0.104,Y -515.699,Z 1734.538,A 0.000,B 0.000,C 90.000,E1 96.834} C_DIS
LIN {X -0.035,Y -516.320,Z 1734.535,A 0.000,B 0.000,C 90.000,E1 96.372} C_DIS
LIN {X -0.167,Y -515.918,Z 1734.533,A 0.000,B 0.000,C 90.000,E1 95.910} C_DIS
LIN {X 0.217,Y -514.429,Z 1734.530,A 0.000,B 0.000,C 90.000,E1 95.391} C_DIS
LIN {X 0.128,Y -513.193,Z 1734.529,A 0.000,B 0.000,C 90.000,E1 95.163} C_DIS
LIN {X -0.104,Y -507.925,Z 1734.525,A 0.000,B 0.000,C 90.000,E1 94.473} C_DIS
LIN {X 0.178,Y -495.365,Z 1734.515,A 0.000,B 0.000,C 90.000,E1 92.751} C_DIS
LIN {X 0.185,Y -482.573,Z 1734.506,A 0.000,B 0.000,C 90.000,E1 91.031} C_DIS
LIN {X -0.067,Y -469.810,Z 1734.496,A 0.000,B 0.000,C 90.000,E1 89.312} C_DIS
LIN {X -0.080,Y -457.004,Z 1734.486,A 0.000,B 0.000,C 90.000,E1 87.535} C_DIS
LIN {X 0.118,Y -444.106,Z 1734.476,A 0.000,B 0.000,C 90.000,E1 85.698} C_DIS
LIN {X 0.093,Y -431.310,Z 1734.466,A 0.000,B 0.000,C 90.000,E1 83.856} C_DIS
LIN {X -0.051,Y -416.889,Z 1734.454,A 0.000,B 0.000,C 90.000,E1 81.724} C_DIS
LIN {X -0.123,Y -397.959,Z 1734.437,A 0.000,B 0.000,C 90.000,E1 78.701} C_DIS
LIN {X 0.141,Y -383.433,Z 1734.423,A 0.000,B 0.000,C 90.000,E1 76.117} C_DIS
LIN {X 0.200,Y -370.940,Z 1734.410,A 0.000,B 0.000,C 90.000,E1 73.795} C_DIS
LIN {X 0.071,Y -358.712,Z 1734.397,A 0.000,B 0.000,C 90.000,E1 71.456} C_DIS
LIN {X -0.065,Y -344.065,Z 1734.380,A 0.000,B 0.000,C 90.000,E1 68.465} C_DIS
LIN {X -0.026,Y -334.275,Z 1734.368,A 0.000,B 0.000,C 90.000,E1 66.305} C_DIS
LIN {X 0.108,Y -321.733,Z 1734.353,A 0.000,B 0.000,C 90.000,E1 63.461} C_DIS
LIN {X 0.010,Y -313.589,Z 1734.342,A 0.000,B 0.000,C 90.000,E1 61.563} C_DIS
LIN {X 0.074,Y -303.872,Z 1734.329,A 0.000,B 0.000,C 90.000,E1 59.282} C_DIS
LIN {X -0.028,Y -294.140,Z 1734.317,A 0.000,B 0.000,C 90.000,E1 56.993} C_DIS
LIN {X 0.004,Y -285.724,Z 1734.305,A 0.000,B 0.000,C 90.000,E1 54.975} C_DIS
LIN {X 0.153,Y -275.922,Z 1734.292,A 0.000,B 0.000,C 90.000,E1 52.557} C_DIS
LIN {X 0.037,Y -266.149,Z 1734.279,A 0.000,B 0.000,C 90.000,E1 50.150} C_DIS
LIN {X 0.062,Y -255.178,Z 1734.263,A 0.000,B 0.000,C 90.000,E1 47.310} C_DIS
LIN {X -0.016,Y -244.654,Z 1734.247,A 0.000,B 0.000,C 90.000,E1 44.433} C_DIS
LIN {X 0.128,Y -233.318,Z 1734.228,A 0.000,B 0.000,C 90.000,E1 41.067} C_DIS
LIN {X 0.036,Y -222.808,Z 1734.209,A 0.000,B 0.000,C 90.000,E1 37.684} C_DIS
LIN {X -0.018,Y -214.380,Z 1734.192,A 0.000,B 0.000,C 90.000,E1 34.612} C_DIS
LIN {X 0.018,Y -206.720,Z 1734.175,A 0.000,B 0.000,C 90.000,E1 31.465} C_DIS
LIN {X -0.002,Y -199.779,Z 1734.157,A 0.000,B 0.000,C 90.000,E1 28.281} C_DIS
LIN {X 0.055,Y -193.564,Z 1734.139,A 0.000,B 0.000,C 90.000,E1 25.027} C_DIS
LIN {X -0.025,Y -187.982,Z 1734.121,A 0.000,B 0.000,C 90.000,E1 21.770} C_DIS
LIN {X 0.072,Y -183.196,Z 1734.102,A 0.000,B 0.000,C 90.000,E1 18.417} C_DIS
LIN {X 0.053,Y -179.113,Z 1734.084,A 0.000,B 0.000,C 90.000,E1 15.064} C_DIS
LIN {X -0.069,Y -175.817,Z 1734.065,A 0.000,B 0.000,C 90.000,E1 11.715} C_DIS
LIN {X 0.035,Y -172.696,Z 1734.041,A 0.000,B 0.000,C 90.000,E1 7.409} C_DIS
LIN {X 0.063,Y -170.163,Z 1734.013,A 0.000,B 0.000,C 90.000,E1 2.236} C_DIS
LIN {X 0.066,Y -169.149,Z 1733.973,A 0.000,B 0.000,C 90.000,E1 355.179} C_DIS
LIN {X -0.064,Y -170.852,Z 1733.920,A 0.000,B 0.000,C 90.000,E1 345.700} C_DIS
LIN {X 0.035,Y -173.502,Z 1733.892,A 0.000,B 0.000,C 90.000,E1 340.496} C_DIS
LIN {X -0.009,Y -176.883,Z 1733.868,A 0.000,B 0.000,C 90.000,E1 336.230} C_DIS
LIN {X 0.018,Y -181.066,Z 1733.844,A 0.000,B 0.000,C 90.000,E1 331.975} C_DIS
LIN {X 0.000,Y -185.327,Z 1733.826,A 0.000,B 0.000,C 90.000,E1 328.614} C_DIS
LIN {X 0.064,Y -190.488,Z 1733.807,A 0.000,B 0.000,C 90.000,E1 325.261} C_DIS
LIN {X 0.029,Y -195.071,Z 1733.793,A 0.000,B 0.000,C 90.000,E1 322.798} C_DIS
LIN {X 0.020,Y -202.265,Z 1733.775,A 0.000,B 0.000,C 90.000,E1 319.542} C_DIS
LIN {X 0.001,Y -209.562,Z 1733.760,A 0.000,B 0.000,C 90.000,E1 316.743} C_DIS
LIN {X 0.095,Y -216.601,Z 1733.747,A 0.000,B 0.000,C 90.000,E1 314.352} C_DIS
LIN {X -0.061,Y -223.227,Z 1733.736,A 0.000,B 0.000,C 90.000,E1 312.447} C_DIS
LIN {X -0.099,Y -230.645,Z 1733.725,A 0.000,B 0.000,C 90.000,E1 310.539} C_DIS
LIN {X 0.009,Y -238.957,Z 1733.715,A 0.000,B 0.000,C 90.000,E1 308.624} C_DIS
LIN {X -0.081,Y -248.240,Z 1733.704,A 0.000,B 0.000,C 90.000,E1 306.790} C_DIS
LIN {X 0.019,Y -258.467,Z 1733.694,A 0.000,B 0.000,C 90.000,E1 304.945} C_DIS
LIN {X -0.101,Y -276.483,Z 1733.678,A 0.000,B 0.000,C 90.000,E1 302.133} C_DIS
LIN {X 0.060,Y -296.108,Z 1733.663,A 0.000,B 0.000,C 90.000,E1 299.361} C_DIS
LIN {X 0.028,Y -314.165,Z 1733.650,A 0.000,B 0.000,C 90.000,E1 297.052} C_DIS
LIN {X -0.073,Y -327.387,Z 1733.641,A 0.000,B 0.000,C 90.000,E1 295.463} C_DIS
LIN {X 0.015,Y -343.235,Z 1733.631,A 0.000,B 0.000,C 90.000,E1 293.567} C_DIS
LIN {X 0.063,Y -353.510,Z 1733.624,A 0.000,B 0.000,C 90.000,E1 292.333} C_DIS
LIN {X -0.035,Y -365.903,Z 1733.616,A 0.000,B 0.000,C 90.000,E1 290.844} C_DIS
LIN {X 0.067,Y -373.025,Z 1733.611,A 0.000,B 0.000,C 90.000,E1 289.939} C_DIS
LIN {X -0.107,Y -379.544,Z 1733.606,A 0.000,B 0.000,C 90.000,E1 289.087} C_DIS
LIN {X 0.009,Y -383.343,Z 1733.603,A 0.000,B 0.000,C 90.000,E1 288.489} C_DIS
LIN {X -0.095,Y -386.767,Z 1733.599,A 0.000,B 0.000,C 90.000,E1 287.928} C_DIS
LIN {X 0.068,Y -389.719,Z 1733.596,A 0.000,B 0.000,C 90.000,E1 287.330} C_DIS
LIN {X -0.235,Y -392.240,Z 1733.593,A 0.000,B 0.000,C 90.000,E1 286.804} C_DIS
LIN {X 0.131,Y -395.209,Z 1733.588,A 0.000,B 0.000,C 90.000,E1 285.898} C_DIS
LIN {X -0.137,Y -396.782,Z 1733.585,A 0.000,B 0.000,C 90.000,E1 285.371} C_DIS
LIN {X 0.094,Y -398.020,Z 1733.582,A 0.000,B 0.000,C 90.000,E1 284.773} C_DIS
LIN {X -0.152,Y -398.874,Z 1733.579,A 0.000,B 0.000,C 90.000,E1 284.245} C_DIS
LIN {X 0.093,Y -399.364,Z 1733.576,A 0.000,B 0.000,C 90.000,E1 283.647} C_DIS
LIN {X -0.139,Y -399.515,Z 1733.573,A 0.000,B 0.000,C 90.000,E1 283.119} C_DIS
LIN {X 0.021,Y -399.280,Z 1733.570,A 0.000,B 0.000,C 90.000,E1 282.535} C_DIS
LIN {X -0.206,Y -398.592,Z 1733.567,A 0.000,B 0.000,C 90.000,E1 282.007} C_DIS
LIN {X -0.044,Y -397.401,Z 1733.563,A 0.000,B 0.000,C 90.000,E1 281.422} C_DIS
LIN {X 0.112,Y -395.704,Z 1733.560,A 0.000,B 0.000,C 90.000,E1 280.838} C_DIS
LIN {X -0.127,Y -393.429,Z 1733.557,A 0.000,B 0.000,C 90.000,E1 280.310} C_DIS
LIN {X -0.007,Y -388.958,Z 1733.552,A 0.000,B 0.000,C 90.000,E1 279.443} C_DIS
LIN {X 0.174,Y -382.289,Z 1733.546,A 0.000,B 0.000,C 90.000,E1 278.276} C_DIS
LIN {X 0.198,Y -377.480,Z 1733.541,A 0.000,B 0.000,C 90.000,E1 277.409} C_DIS
LIN {X 0.173,Y -373.781,Z 1733.538,A 0.000,B 0.000,C 90.000,E1 276.834} C_DIS
LIN {X 0.129,Y -369.467,Z 1733.535,A 0.000,B 0.000,C 90.000,E1 276.258} C_DIS
LIN {X 0.064,Y -364.490,Z 1733.532,A 0.000,B 0.000,C 90.000,E1 275.682} C_DIS
LIN {X 0.000,Y -358.806,Z 1733.528,A 0.000,B 0.000,C 90.000,E1 275.106} C_DIS
LIN {X -0.145,Y -352.888,Z 1733.525,A 0.000,B 0.000,C 90.000,E1 274.588} C_DIS
LIN {X -0.086,Y -346.875,Z 1733.523,A 0.000,B 0.000,C 90.000,E1 274.073} C_DIS
LIN {X -0.052,Y -337.587,Z 1733.519,A 0.000,B 0.000,C 90.000,E1 273.383} C_DIS
LIN {X -0.100,Y -331.247,Z 1733.516,A 0.000,B 0.000,C 90.000,E1 272.980} C_DIS
LIN {X 0.062,Y -324.760,Z 1733.514,A 0.000,B 0.000,C 90.000,E1 272.579} C_DIS
LIN {X 0.115,Y -318.232,Z 1733.513,A 0.000,B 0.000,C 90.000,E1 272.236} C_DIS
LIN {X 0.076,Y -311.400,Z 1733.511,A 0.000,B 0.000,C 90.000,E1 271.949} C_DIS
LIN {X -0.030,Y -304.477,Z 1733.510,A 0.000,B 0.000,C 90.000,E1 271.718} C_DIS
LIN {X 0.106,Y -293.464,Z 1733.508,A 0.000,B 0.000,C 90.000,E1 271.375} C_DIS
LIN {X 0.034,Y -281.891,Z 1733.506,A 0.000,B 0.000,C 90.000,E1 271.146} C_DIS
LIN {X -0.055,Y -269.050,Z 1733.505,A 0.000,B 0.000,C 90.000,E1 270.974} C_DIS
LIN {X -0.013,Y -253.608,Z 1733.504,A 0.000,B 0.000,C 90.000,E1 270.802} C_DIS
LIN {X -0.078,Y -241.711,Z 1733.504,A 0.000,B 0.000,C 90.000,E1 270.745} C_DIS
LIN {X 0.115,Y -234.963,Z 1733.504,A 0.000,B 0.000,C 90.000,E1 270.688} C_DIS
LIN {X 0.054,Y -181.525,Z 1733.504,A 0.000,B 0.000,C 90.000,E1 270.688} C_DIS
LIN {X -0.028,Y -181.523,Z 1733.499,A 0.000,B 0.000,C 90.000,E1 269.828} C_DIS
LIN {X -0.044,Y -180.793,Z 1733.471,A 0.000,B 0.000,C 90.000,E1 264.780} C_DIS
LIN {X 0.029,Y -178.891,Z 1733.443,A 0.000,B 0.000,C 90.000,E1 259.690} C_DIS
LIN {X -0.066,Y -175.934,Z 1733.414,A 0.000,B 0.000,C 90.000,E1 254.629} C_DIS
LIN {X 0.050,Y -175.382,Z 1733.410,A 0.000,B 0.000,C 90.000,E1 253.740} C_DIS
LIN {X 0.047,Y -172.155,Z 1733.386,A 0.000,B 0.000,C 90.000,E1 249.464} C_DIS
LIN {X 0.085,Y -171.622,Z 1733.381,A 0.000,B 0.000,C 90.000,E1 248.592} C_DIS
LIN {X 0.072,Y -167.844,Z 1733.357,A 0.000,B 0.000,C 90.000,E1 244.280} C_DIS
LIN {X 0.013,Y -166.573,Z 1733.348,A 0.000,B 0.000,C 90.000,E1 242.564} C_DIS
LIN {X -0.001,Y -162.565,Z 1733.323,A 0.000,B 0.000,C 90.000,E1 238.201} C_DIS
LIN {X 0.059,Y -161.246,Z 1733.314,A 0.000,B 0.000,C 90.000,E1 236.421} C_DIS
LIN {X -0.031,Y -157.249,Z 1733.289,A 0.000,B 0.000,C 90.000,E1 232.029} C_DIS
LIN {X 0.016,Y -155.972,Z 1733.279,A 0.000,B 0.000,C 90.000,E1 230.231} C_DIS
LIN {X 0.073,Y -152.227,Z 1733.254,A 0.000,B 0.000,C 90.000,E1 225.729} C_DIS
LIN {X -0.017,Y -150.470,Z 1733.239,A 0.000,B 0.000,C 90.000,E1 223.056} C_DIS
LIN {X 0.003,Y -147.194,Z 1733.214,A 0.000,B 0.000,C 90.000,E1 218.508} C_DIS
LIN {X 0.085,Y -145.213,Z 1733.194,A 0.000,B 0.000,C 90.000,E1 214.818} C_DIS
LIN {X -0.006,Y -142.345,Z 1733.163,A 0.000,B 0.000,C 90.000,E1 209.333} C_DIS
LIN {X 0.047,Y -141.733,Z 1733.153,A 0.000,B 0.000,C 90.000,E1 207.462} C_DIS
LIN {X 0.029,Y -139.484,Z 1733.117,A 0.000,B 0.000,C 90.000,E1 200.972} C_DIS
LIN {X 0.018,Y -138.985,Z 1733.101,A 0.000,B 0.000,C 90.000,E1 198.181} C_DIS
LIN {X -0.021,Y -138.334,Z 1733.054,A 0.000,B 0.000,C 90.000,E1 189.792} C_DIS
LIN {X 0.003,Y -139.425,Z 1733.008,A 0.000,B 0.000,C 90.000,E1 181.375} C_DIS
LIN {X 0.058,Y -141.348,Z 1732.971,A 0.000,B 0.000,C 90.000,E1 174.837} C_DIS
LIN {X 0.034,Y -142.703,Z 1732.956,A 0.000,B 0.000,C 90.000,E1 172.064} C_DIS
LIN {X -0.007,Y -145.073,Z 1732.930,A 0.000,B 0.000,C 90.000,E1 167.465} C_DIS
LIN {X -0.010,Y -147.698,Z 1732.910,A 0.000,B 0.000,C 90.000,E1 163.795} C_DIS
LIN {X 0.023,Y -150.349,Z 1732.890,A 0.000,B 0.000,C 90.000,E1 160.134} C_DIS
LIN {X 0.016,Y -154.603,Z 1732.865,A 0.000,B 0.000,C 90.000,E1 155.613} C_DIS
LIN {X 0.023,Y -158.145,Z 1732.845,A 0.000,B 0.000,C 90.000,E1 152.025} C_DIS
LIN {X 0.067,Y -162.430,Z 1732.825,A 0.000,B 0.000,C 90.000,E1 148.456} C_DIS
LIN {X -0.036,Y -166.690,Z 1732.805,A 0.000,B 0.000,C 90.000,E1 144.975} C_DIS
LIN {X 0.076,Y -171.695,Z 1732.786,A 0.000,B 0.000,C 90.000,E1 141.457} C_DIS
LIN {X 0.011,Y -176.668,Z 1732.767,A 0.000,B 0.000,C 90.000,E1 138.038} C_DIS
LIN {X 0.006,Y -180.964,Z 1732.753,A 0.000,B 0.000,C 90.000,E1 135.486} C_DIS
LIN {X -0.007,Y -186.387,Z 1732.734,A 0.000,B 0.000,C 90.000,E1 132.123} C_DIS
LIN {X -0.068,Y -191.017,Z 1732.720,A 0.000,B 0.000,C 90.000,E1 129.644} C_DIS
LIN {X 0.126,Y -196.796,Z 1732.702,A 0.000,B 0.000,C 90.000,E1 126.297} C_DIS
LIN {X 0.045,Y -200.048,Z 1732.693,A 0.000,B 0.000,C 90.000,E1 124.692} C_DIS
LIN {X 0.040,Y -207.549,Z 1732.670,A 0.000,B 0.000,C 90.000,E1 120.669} C_DIS
LIN {X -0.060,Y -209.967,Z 1732.664,A 0.000,B 0.000,C 90.000,E1 119.539} C_DIS
LIN {X -0.162,Y -334.145,Z 1732.664,A 0.000,B 0.000,C 90.000,E1 119.539} C_DIS
LIN {X 0.064,Y -335.446,Z 1732.664,A 0.000,B 0.000,C 90.000,E1 119.489} C_DIS
LIN {X 0.068,Y -340.883,Z 1732.663,A 0.000,B 0.000,C 90.000,E1 119.283} C_DIS
LIN {X 0.070,Y -343.559,Z 1732.662,A 0.000,B 0.000,C 90.000,E1 119.077} C_DIS
LIN {X 0.161,Y -347.331,Z 1732.659,A 0.000,B 0.000,C 90.000,E1 118.615} C_DIS
LIN {X -0.147,Y -349.125,Z 1732.657,A 0.000,B 0.000,C 90.000,E1 118.359} C_DIS
LIN {X -0.126,Y -363.628,Z 1732.641,A 0.000,B 0.000,C 90.000,E1 115.335} C_DIS
LIN {X 0.126,Y -378.243,Z 1732.626,A 0.000,B 0.000,C 90.000,E1 112.642} C_DIS
LIN {X -0.004,Y -392.625,Z 1732.613,A 0.000,B 0.000,C 90.000,E1 110.355} C_DIS
LIN {X -0.064,Y -408.417,Z 1732.601,A 0.000,B 0.000,C 90.000,E1 108.109} C_DIS
LIN {X 0.016,Y -425.731,Z 1732.588,A 0.000,B 0.000,C 90.000,E1 105.898} C_DIS
LIN {X -0.113,Y -444.684,Z 1732.576,A 0.000,B 0.000,C 90.000,E1 103.772} C_DIS
LIN {X -0.211,Y -464.663,Z 1732.565,A 0.000,B 0.000,C 90.000,E1 101.771} C_DIS
LIN {X 0.040,Y -487.776,Z 1732.554,A 0.000,B 0.000,C 90.000,E1 99.670} C_DIS
LIN {X -0.042,Y -508.749,Z 1732.544,A 0.000,B 0.000,C 90.000,E1 97.992} C_DIS
LIN {X 0.248,Y -510.749,Z 1732.543,A 0.000,B 0.000,C 90.000,E1 97.757} C_DIS
LIN {X 0.130,Y -512.543,Z 1732.542,A 0.000,B 0.000,C 90.000,E1 97.530} C_DIS
LIN {X 0.080,Y -513.885,Z 1732.541,A 0.000,B 0.000,C 90.000,E1 97.296} C_DIS
LIN {X -0.066,Y -515.541,Z 1732.538,A 0.000,B 0.000,C 90.000,E1 96.834} C_DIS
LIN {X -0.207,Y -516.087,Z 1732.535,A 0.000,B 0.000,C 90.000,E1 96.372} C_DIS
LIN {X 0.175,Y -515.613,Z 1732.533,A 0.000,B 0.000,C 90.000,E1 95.853} C_DIS
LIN {X 0.045,Y -514.039,Z 1732.530,A 0.000,B 0.000,C 90.000,E1 95.391} C_DIS
LIN {X -0.045,Y -512.750,Z 1732.529,A 0.000,B 0.000,C 90.000,E1 95.163} C_DIS
LIN {X -0.052,Y -502.014,Z 1732.521,A 0.000,B 0.000,C 90.000,E1 93.726} C_DIS
LIN {X 0.228,Y -491.236,Z 1732.513,A 0.000,B 0.000,C 90.000,E1 92.236} C_DIS
LIN {X -0.014,Y -476.579,Z 1732.502,A 0.000,B 0.000,C 90.000,E1 90.286} C_DIS
LIN {X 0.093,Y -463.820,Z 1732.492,A 0.000,B 0.000,C 90.000,E1 88.511} C_DIS
LIN {X -0.029,Y -450.962,Z 1732.482,A 0.000,B 0.000,C 90.000,E1 86.731} C_DIS
LIN {X -0.222,Y -436.265,Z 1732.470,A 0.000,B 0.000,C 90.000,E1 84.666} C_DIS
LIN {X 0.227,Y -421.728,Z 1732.458,A 0.000,B 0.000,C 90.000,E1 82.470} C_DIS
LIN {X -0.151,Y -402.464,Z 1732.442,A 0.000,B 0.000,C 90.000,E1 79.511} C_DIS
LIN {X -0.168,Y -386.067,Z 1732.426,A 0.000,B 0.000,C 90.000,E1 76.700} C_DIS
LIN {X -0.130,Y -373.469,Z 1732.413,A 0.000,B 0.000,C 90.000,E1 74.393} C_DIS
LIN {X 0.154,Y -361.175,Z 1732.400,A 0.000,B 0.000,C 90.000,E1 72.000} C_DIS
LIN {X -0.010,Y -344.944,Z 1732.382,A 0.000,B 0.000,C 90.000,E1 68.720} C_DIS
LIN {X 0.167,Y -333.676,Z 1732.368,A 0.000,B 0.000,C 90.000,E1 66.230} C_DIS
LIN {X -0.002,Y -321.115,Z 1732.352,A 0.000,B 0.000,C 90.000,E1 63.435} C_DIS
LIN {X 0.025,Y -312.941,Z 1732.342,A 0.000,B 0.000,C 90.000,E1 61.513} C_DIS
LIN {X -0.036,Y -303.260,Z 1732.329,A 0.000,B 0.000,C 90.000,E1 59.253} C_DIS
LIN {X 0.109,Y -293.552,Z 1732.316,A 0.000,B 0.000,C 90.000,E1 56.914} C_DIS
LIN {X 0.129,Y -285.158,Z 1732.305,A 0.000,B 0.000,C 90.000,E1 54.895} C_DIS
LIN {X -0.122,Y -275.367,Z 1732.292,A 0.000,B 0.000,C 90.000,E1 52.557} C_DIS
LIN {X -0.071,Y -265.593,Z 1732.278,A 0.000,B 0.000,C 90.000,E1 50.114} C_DIS
LIN {X 0.143,Y -254.625,Z 1732.263,A 0.000,B 0.000,C 90.000,E1 47.229} C_DIS
LIN {X -0.134,Y -242.806,Z 1732.244,A 0.000,B 0.000,C 90.000,E1 44.028} C_DIS
LIN {X 0.140,Y -231.567,Z 1732.226,A 0.000,B 0.000,C 90.000,E1 40.620} C_DIS
LIN {X 0.062,Y -222.301,Z 1732.209,A 0.000,B 0.000,C 90.000,E1 37.604} C_DIS
LIN {X 0.000,Y -213.943,Z 1732.192,A 0.000,B 0.000,C 90.000,E1 34.532} C_DIS
LIN {X 0.021,Y -206.349,Z 1732.174,A 0.000,B 0.000,C 90.000,E1 31.386} C_DIS
LIN {X -0.106,Y -199.455,Z 1732.157,A 0.000,B 0.000,C 90.000,E1 28.231} C_DIS
LIN {X 0.033,Y -193.270,Z 1732.139,A 0.000,B 0.000,C 90.000,E1 24.951} C_DIS
LIN {X 0.046,Y -187.720,Z 1732.120,A 0.000,B 0.000,C 90.000,E1 21.663} C_DIS
LIN {X -0.032,Y -182.968,Z 1732.102,A 0.000,B 0.000,C 90.000,E1 18.362} C_DIS
LIN {X -0.050,Y -178.920,Z 1732.083,A 0.000,B 0.000,C 90.000,E1 15.009} C_DIS
LIN {X 0.035,Y -175.621,Z 1732.064,A 0.000,B 0.000,C 90.000,E1 11.591} C_DIS
LIN {X -0.071,Y -172.516,Z 1732.041,A 0.000,B 0.000,C 90.000,E1 7.352} C_DIS
LIN {X -0.046,Y -169.981,Z 1732.012,A 0.000,B 0.000,C 90.000,E1 2.178} C_DIS
LIN {X 0.046,Y -168.987,Z 1731.969,A 0.000,B 0.000,C 90.000,E1 354.318} C_DIS
LIN {X -0.079,Y -170.727,Z 1731.920,A 0.000,B 0.000,C 90.000,E1 345.700} C_DIS
LIN {X 0.016,Y -173.398,Z 1731.892,A 0.000,B 0.000,C 90.000,E1 340.496} C_DIS
LIN {X -0.032,Y -176.781,Z 1731.868,A 0.000,B 0.000,C 90.000,E1 336.230} C_DIS
LIN {X -0.009,Y -181.018,Z 1731.844,A 0.000,B 0.000,C 90.000,E1 331.975} C_DIS
LIN {X -0.029,Y -185.310,Z 1731.826,A 0.000,B 0.000,C 90.000,E1 328.614} C_DIS
LIN {X 0.034,Y -190.512,Z 1731.807,A 0.000,B 0.000,C 90.000,E1 325.261} C_DIS
LIN {X -0.001,Y -195.106,Z 1731.793,A 0.000,B 0.000,C 90.000,E1 322.798} C_DIS
LIN {X -0.009,Y -202.355,Z 1731.775,A 0.000,B 0.000,C 90.000,E1 319.542} C_DIS
LIN {X -0.028,Y -209.690,Z 1731.760,A 0.000,B 0.000,C 90.000,E1 316.743} C_DIS
LIN {X 0.068,Y -216.776,Z 1731.746,A 0.000,B 0.000,C 90.000,E1 314.352} C_DIS
LIN {X -0.010,Y -224.836,Z 1731.734,A 0.000,B 0.000,C 90.000,E1 312.043} C_DIS
LIN {X -0.029,Y -232.417,Z 1731.723,A 0.000,B 0.000,C 90.000,E1 310.135} C_DIS
LIN {X -0.038,Y -240.890,Z 1731.713,A 0.000,B 0.000,C 90.000,E1 308.257} C_DIS
LIN {X 0.096,Y -250.355,Z 1731.702,A 0.000,B 0.000,C 90.000,E1 306.377} C_DIS
LIN {X -0.117,Y -260.823,Z 1731.692,A 0.000,B 0.000,C 90.000,E1 304.612} C_DIS
LIN {X 0.059,Y -279.082,Z 1731.677,A 0.000,B 0.000,C 90.000,E1 301.750} C_DIS
LIN {X 0.053,Y -298.870,Z 1731.661,A 0.000,B 0.000,C 90.000,E1 299.027} C_DIS
LIN {X -0.059,Y -316.999,Z 1731.649,A 0.000,B 0.000,C 90.000,E1 296.744} C_DIS
LIN {X -0.128,Y -330.198,Z 1731.640,A 0.000,B 0.000,C 90.000,E1 295.155} C_DIS
LIN {X 0.002,Y -343.434,Z 1731.631,A 0.000,B 0.000,C 90.000,E1 293.567} C_DIS
LIN {X 0.046,Y -353.703,Z 1731.624,A 0.000,B 0.000,C 90.000,E1 292.333} C_DIS
LIN {X -0.049,Y -366.103,Z 1731.616,A 0.000,B 0.000,C 90.000,E1 290.844} C_DIS
LIN {X 0.055,Y -373.220,Z 1731.611,A 0.000,B 0.000,C 90.000,E1 289.939} C_DIS
LIN {X -0.117,Y -379.758,Z 1731.606,A 0.000,B 0.000,C 90.000,E1 289.087} C_DIS
LIN {X -0.001,Y -383.548,Z 1731.603,A 0.000,B 0.000,C 90.000,E1 288.489} C_DIS
LIN {X -0.104,Y -386.982,Z 1731.599,A 0.000,B 0.000,C 90.000,E1 287.928} C_DIS
LIN {X 0.060,Y -389.925,Z 1731.596,A 0.000,B 0.000,C 90.000,E1 287.330} C_DIS
LIN {X -0.241,Y -392.417,Z 1731.593,A 0.000,B 0.000,C 90.000,E1 286.804} C_DIS
LIN {X 0.127,Y -395.459,Z 1731.588,A 0.000,B 0.000,C 90.000,E1 285.898} C_DIS
LIN {X -0.140,Y -397.026,Z 1731.585,A 0.000,B 0.000,C 90.000,E1 285.371} C_DIS
LIN {X 0.092,Y -398.250,Z 1731.582,A 0.000,B 0.000,C 90.000,E1 284.773} C_DIS
LIN {X -0.152,Y -399.132,Z 1731.579,A 0.000,B 0.000,C 90.000,E1 284.245} C_DIS
LIN {X 0.095,Y -399.602,Z 1731.576,A 0.000,B 0.000,C 90.000,E1 283.647} C_DIS
LIN {X -0.136,Y -399.754,Z 1731.573,A 0.000,B 0.000,C 90.000,E1 283.119} C_DIS
LIN {X 0.025,Y -399.502,Z 1731.570,A 0.000,B 0.000,C 90.000,E1 282.535} C_DIS
LIN {X -0.200,Y -398.810,Z 1731.567,A 0.000,B 0.000,C 90.000,E1 282.007} C_DIS
LIN {X -0.037,Y -397.630,Z 1731.563,A 0.000,B 0.000,C 90.000,E1 281.422} C_DIS
LIN {X 0.120,Y -395.911,Z 1731.560,A 0.000,B 0.000,C 90.000,E1 280.838} C_DIS
LIN {X -0.118,Y -393.634,Z 1731.557,A 0.000,B 0.000,C 90.000,E1 280.310} C_DIS
LIN {X 0.013,Y -390.789,Z 1731.554,A 0.000,B 0.000,C 90.000,E1 279.726} C_DIS
LIN {X 0.192,Y -379.327,Z 1731.543,A 0.000,B 0.000,C 90.000,E1 277.701} C_DIS
LIN {X -0.194,Y -375.832,Z 1731.540,A 0.000,B 0.000,C 90.000,E1 277.182} C_DIS
LIN {X 0.148,Y -371.789,Z 1731.536,A 0.000,B 0.000,C 90.000,E1 276.549} C_DIS
LIN {X 0.133,Y -367.178,Z 1731.533,A 0.000,B 0.000,C 90.000,E1 275.967} C_DIS
LIN {X 0.056,Y -361.791,Z 1731.530,A 0.000,B 0.000,C 90.000,E1 275.391} C_DIS
LIN {X 0.099,Y -355.931,Z 1731.527,A 0.000,B 0.000,C 90.000,E1 274.821} C_DIS
LIN {X 0.087,Y -349.997,Z 1731.524,A 0.000,B 0.000,C 90.000,E1 274.302} C_DIS
LIN {X -0.054,Y -343.914,Z 1731.521,A 0.000,B 0.000,C 90.000,E1 273.841} C_DIS
LIN {X 0.020,Y -337.699,Z 1731.519,A 0.000,B 0.000,C 90.000,E1 273.383} C_DIS
LIN {X -0.015,Y -331.363,Z 1731.516,A 0.000,B 0.000,C 90.000,E1 272.980} C_DIS
LIN {X 0.128,Y -324.736,Z 1731.514,A 0.000,B 0.000,C 90.000,E1 272.579} C_DIS
LIN {X -0.157,Y -318.067,Z 1731.513,A 0.000,B 0.000,C 90.000,E1 272.293} C_DIS
LIN {X 0.109,Y -311.180,Z 1731.511,A 0.000,B 0.000,C 90.000,E1 271.949} C_DIS
LIN {X -0.006,Y -304.102,Z 1731.510,A 0.000,B 0.000,C 90.000,E1 271.718} C_DIS
LIN {X 0.146,Y -292.987,Z 1731.508,A 0.000,B 0.000,C 90.000,E1 271.375} C_DIS
LIN {X 0.098,Y -281.623,Z 1731.506,A 0.000,B 0.000,C 90.000,E1 271.146} C_DIS
LIN {X 0.028,Y -269.027,Z 1731.505,A 0.000,B 0.000,C 90.000,E1 270.974} C_DIS
LIN {X 0.059,Y -253.362,Z 1731.505,A 0.000,B 0.000,C 90.000,E1 270.802} C_DIS
LIN {X -0.005,Y -237.974,Z 1731.504,A 0.000,B 0.000,C 90.000,E1 270.745} C_DIS
LIN {X -0.038,Y -181.518,Z 1731.504,A 0.000,B 0.000,C 90.000,E1 270.745} C_DIS
LIN {X 0.032,Y -181.528,Z 1731.499,A 0.000,B 0.000,C 90.000,E1 269.828} C_DIS
LIN {X 0.015,Y -180.800,Z 1731.471,A 0.000,B 0.000,C 90.000,E1 264.780} C_DIS
LIN {X -0.087,Y -178.900,Z 1731.443,A 0.000,B 0.000,C 90.000,E1 259.746} C_DIS
LIN {X -0.006,Y -175.943,Z 1731.415,A 0.000,B 0.000,C 90.000,E1 254.629} C_DIS
LIN {X -0.059,Y -175.399,Z 1731.410,A 0.000,B 0.000,C 90.000,E1 253.795} C_DIS
LIN {X -0.056,Y -172.167,Z 1731.386,A 0.000,B 0.000,C 90.000,E1 249.518} C_DIS
LIN {X -0.017,Y -171.635,Z 1731.381,A 0.000,B 0.000,C 90.000,E1 248.646} C_DIS
LIN {X -0.022,Y -167.859,Z 1731.357,A 0.000,B 0.000,C 90.000,E1 244.332} C_DIS
LIN {X -0.078,Y -166.591,Z 1731.348,A 0.000,B 0.000,C 90.000,E1 242.615} C_DIS
LIN {X 0.055,Y -162.581,Z 1731.323,A 0.000,B 0.000,C 90.000,E1 238.201} C_DIS
LIN {X -0.109,Y -161.264,Z 1731.314,A 0.000,B 0.000,C 90.000,E1 236.501} C_DIS
LIN {X 0.024,Y -157.265,Z 1731.289,A 0.000,B 0.000,C 90.000,E1 232.029} C_DIS
LIN {X -0.050,Y -155.985,Z 1731.279,A 0.000,B 0.000,C 90.000,E1 230.275} C_DIS
LIN {X -0.088,Y -152.241,Z 1731.254,A 0.000,B 0.000,C 90.000,E1 225.810} C_DIS
LIN {X 0.037,Y -150.483,Z 1731.239,A 0.000,B 0.000,C 90.000,E1 223.056} C_DIS
LIN {X -0.035,Y -147.208,Z 1731.214,A 0.000,B 0.000,C 90.000,E1 218.543} C_DIS
LIN {X -0.065,Y -145.227,Z 1731.194,A 0.000,B 0.000,C 90.000,E1 214.898} C_DIS
LIN {X 0.047,Y -142.353,Z 1731.163,A 0.000,B 0.000,C 90.000,E1 209.333} C_DIS
LIN {X -0.026,Y -141.741,Z 1731.153,A 0.000,B 0.000,C 90.000,E1 207.513} C_DIS
LIN {X 0.081,Y -139.488,Z 1731.117,A 0.000,B 0.000,C 90.000,E1 200.972} C_DIS
LIN {X 0.069,Y -138.990,Z 1731.101,A 0.000,B 0.000,C 90.000,E1 198.181} C_DIS
LIN {X 0.030,Y -138.335,Z 1731.054,A 0.000,B 0.000,C 90.000,E1 189.792} C_DIS
LIN {X 0.055,Y -139.419,Z 1731.008,A 0.000,B 0.000,C 90.000,E1 181.375} C_DIS
LIN {X -0.032,Y -141.339,Z 1730.972,A 0.000,B 0.000,C 90.000,E1 174.894} C_DIS
LIN {X -0.075,Y -142.695,Z 1730.956,A 0.000,B 0.000,C 90.000,E1 172.129} C_DIS
LIN {X 0.046,Y -145.060,Z 1730.930,A 0.000,B 0.000,C 90.000,E1 167.465} C_DIS
LIN {X 0.042,Y -147.685,Z 1730.910,A 0.000,B 0.000,C 90.000,E1 163.795} C_DIS
LIN {X -0.065,Y -150.332,Z 1730.890,A 0.000,B 0.000,C 90.000,E1 160.188} C_DIS
LIN {X 0.006,Y -153.750,Z 1730.870,A 0.000,B 0.000,C 90.000,E1 156.538} C_DIS
LIN {X -0.003,Y -157.162,Z 1730.850,A 0.000,B 0.000,C 90.000,E1 152.948} C_DIS
LIN {X -0.069,Y -161.316,Z 1730.830,A 0.000,B 0.000,C 90.000,E1 149.410} C_DIS
LIN {X -0.053,Y -164.430,Z 1730.815,A 0.000,B 0.000,C 90.000,E1 146.755} C_DIS
LIN {X 0.079,Y -169.116,Z 1730.796,A 0.000,B 0.000,C 90.000,E1 143.210} C_DIS
LIN {X -0.106,Y -171.670,Z 1730.786,A 0.000,B 0.000,C 90.000,E1 141.537} C_DIS
LIN {X -0.061,Y -176.637,Z 1730.767,A 0.000,B 0.000,C 90.000,E1 138.081} C_DIS
LIN {X 0.067,Y -180.934,Z 1730.753,A 0.000,B 0.000,C 90.000,E1 135.486} C_DIS
LIN {X 0.055,Y -186.354,Z 1730.734,A 0.000,B 0.000,C 90.000,E1 132.123} C_DIS
LIN {X -0.004,Y -190.986,Z 1730.720,A 0.000,B 0.000,C 90.000,E1 129.644} C_DIS
LIN {X -0.086,Y -196.761,Z 1730.702,A 0.000,B 0.000,C 90.000,E1 126.377} C_DIS
LIN {X -0.055,Y -200.010,Z 1730.693,A 0.000,B 0.000,C 90.000,E1 124.739} C_DIS
LIN {X -0.074,Y -207.512,Z 1730.671,A 0.000,B 0.000,C 90.000,E1 120.718} C_DIS
LIN {X 0.047,Y -209.908,Z 1730.664,A 0.000,B 0.000,C 90.000,E1 119.539} C_DIS
LIN {X 0.009,Y -334.384,Z 1730.664,A 0.000,B 0.000,C 90.000,E1 119.539} C_DIS
LIN {X -0.122,Y -336.044,Z 1730.664,A 0.000,B 0.000,C 90.000,E1 119.539} C_DIS
LIN {X -0.122,Y -340.928,Z 1730.663,A 0.000,B 0.000,C 90.000,E1 119.333} C_DIS
LIN {X 0.178,Y -343.538,Z 1730.662,A 0.000,B 0.000,C 90.000,E1 119.077} C_DIS
LIN {X 0.213,Y -347.317,Z 1730.659,A 0.000,B 0.000,C 90.000,E1 118.615} C_DIS
LIN {X -0.095,Y -349.078,Z 1730.657,A 0.000,B 0.000,C 90.000,E1 118.359} C_DIS
LIN {X -0.074,Y -363.562,Z 1730.641,A 0.000,B 0.000,C 90.000,E1 115.335} C_DIS
LIN {X 0.179,Y -378.172,Z 1730.626,A 0.000,B 0.000,C 90.000,E1 112.642} C_DIS
LIN {X 0.050,Y -392.549,Z 1730.613,A 0.000,B 0.000,C 90.000,E1 110.355} C_DIS
LIN {X -0.137,Y -408.336,Z 1730.601,A 0.000,B 0.000,C 90.000,E1 108.127} C_DIS
LIN {X 0.070,Y -425.643,Z 1730.588,A 0.000,B 0.000,C 90.000,E1 105.898} C_DIS
LIN {X -0.060,Y -444.591,Z 1730.576,A 0.000,B 0.000,C 90.000,E1 103.772} C_DIS
LIN {X -0.160,Y -464.568,Z 1730.565,A 0.000,B 0.000,C 90.000,E1 101.771} C_DIS
LIN {X 0.087,Y -487.679,Z 1730.554,A 0.000,B 0.000,C 90.000,E1 99.670} C_DIS
LIN {X 0.003,Y -508.632,Z 1730.544,A 0.000,B 0.000,C 90.000,E1 97.992} C_DIS
LIN {X -0.214,Y -510.602,Z 1730.543,A 0.000,B 0.000,C 90.000,E1 97.814} C_DIS
LIN {X 0.175,Y -512.373,Z 1730.542,A 0.000,B 0.000,C 90.000,E1 97.530} C_DIS
LIN {X 0.125,Y -513.696,Z 1730.541,A 0.000,B 0.000,C 90.000,E1 97.296} C_DIS
LIN {X -0.023,Y -515.324,Z 1730.538,A 0.000,B 0.000,C 90.000,E1 96.834} C_DIS
LIN {X -0.164,Y -515.848,Z 1730.535,A 0.000,B 0.000,C 90.000,E1 96.372} C_DIS
LIN {X 0.215,Y -515.354,Z 1730.533,A 0.000,B 0.000,C 90.000,E1 95.853} C_DIS
LIN {X 0.084,Y -513.754,Z 1730.530,A 0.000,B 0.000,C 90.000,E1 95.391} C_DIS
LIN {X -0.006,Y -512.448,Z 1730.529,A 0.000,B 0.000,C 90.000,E1 95.163} C_DIS
LIN {X -0.130,Y -499.894,Z 1730.519,A 0.000,B 0.000,C 90.000,E1 93.498} C_DIS
LIN {X 0.118,Y -489.085,Z 1730.511,A 0.000,B 0.000,C 90.000,E1 92.007} C_DIS
LIN {X -0.166,Y -474.455,Z 1730.500,A 0.000,B 0.000,C 90.000,E1 90.057} C_DIS
LIN {X -0.104,Y -461.647,Z 1730.490,A 0.000,B 0.000,C 90.000,E1 88.282} C_DIS
LIN {X 0.189,Y -448.786,Z 1730.480,A 0.000,B 0.000,C 90.000,E1 86.445} C_DIS
LIN {X -0.226,Y -435.933,Z 1730.470,A 0.000,B 0.000,C 90.000,E1 84.666} C_DIS
LIN {X 0.216,Y -421.361,Z 1730.458,A 0.000,B 0.000,C 90.000,E1 82.470} C_DIS
LIN {X -0.173,Y -402.087,Z 1730.442,A 0.000,B 0.000,C 90.000,E1 79.511} C_DIS
LIN {X 0.175,Y -385.685,Z 1730.426,A 0.000,B 0.000,C 90.000,E1 76.645} C_DIS
LIN {X -0.170,Y -373.072,Z 1730.413,A 0.000,B 0.000,C 90.000,E1 74.393} C_DIS
LIN {X 0.106,Y -360.760,Z 1730.400,A 0.000,B 0.000,C 90.000,E1 72.000} C_DIS
LIN {X -0.070,Y -344.534,Z 1730.382,A 0.000,B 0.000,C 90.000,E1 68.720} C_DIS
LIN {X 0.099,Y -333.213,Z 1730.368,A 0.000,B 0.000,C 90.000,E1 66.230} C_DIS
LIN {X -0.081,Y -320.629,Z 1730.352,A 0.000,B 0.000,C 90.000,E1 63.435} C_DIS
LIN {X -0.060,Y -312.429,Z 1730.342,A 0.000,B 0.000,C 90.000,E1 61.513} C_DIS
LIN {X 0.131,Y -302.784,Z 1730.329,A 0.000,B 0.000,C 90.000,E1 59.203} C_DIS
LIN {X 0.008,Y -293.104,Z 1730.316,A 0.000,B 0.000,C 90.000,E1 56.914} C_DIS
LIN {X 0.023,Y -284.733,Z 1730.305,A 0.000,B 0.000,C 90.000,E1 54.895} C_DIS
LIN {X 0.152,Y -274.949,Z 1730.292,A 0.000,B 0.000,C 90.000,E1 52.477} C_DIS
LIN {X 0.016,Y -265.172,Z 1730.278,A 0.000,B 0.000,C 90.000,E1 50.070} C_DIS
LIN {X -0.016,Y -255.567,Z 1730.264,A 0.000,B 0.000,C 90.000,E1 47.595} C_DIS
LIN {X -0.080,Y -243.653,Z 1730.246,A 0.000,B 0.000,C 90.000,E1 44.352} C_DIS
LIN {X 0.039,Y -232.359,Z 1730.228,A 0.000,B 0.000,C 90.000,E1 40.987} C_DIS
LIN {X -0.077,Y -221.922,Z 1730.209,A 0.000,B 0.000,C 90.000,E1 37.604} C_DIS
LIN {X 0.033,Y -213.612,Z 1730.192,A 0.000,B 0.000,C 90.000,E1 34.485} C_DIS
LIN {X 0.051,Y -206.078,Z 1730.174,A 0.000,B 0.000,C 90.000,E1 31.337} C_DIS
LIN {X 0.016,Y -199.227,Z 1730.156,A 0.000,B 0.000,C 90.000,E1 28.153} C_DIS
LIN {X 0.060,Y -193.062,Z 1730.138,A 0.000,B 0.000,C 90.000,E1 24.899} C_DIS
LIN {X -0.033,Y -187.530,Z 1730.120,A 0.000,B 0.000,C 90.000,E1 21.642} C_DIS
LIN {X -0.007,Y -182.789,Z 1730.102,A 0.000,B 0.000,C 90.000,E1 18.308} C_DIS
LIN {X -0.028,Y -178.783,Z 1730.083,A 0.000,B 0.000,C 90.000,E1 14.954} C_DIS
LIN {X -0.042,Y -174.765,Z 1730.059,A 0.000,B 0.000,C 90.000,E1 10.715} C_DIS
LIN {X -0.025,Y -171.345,Z 1730.031,A 0.000,B 0.000,C 90.000,E1 5.568} C_DIS
LIN {X -0.030,Y -169.195,Z 1729.997,A 0.000,B 0.000,C 90.000,E1 359.542} C_DIS
LIN {X 0.022,Y -168.867,Z 1729.964,A 0.000,B 0.000,C 90.000,E1 353.457} C_DIS
LIN {X 0.072,Y -170.599,Z 1729.920,A 0.000,B 0.000,C 90.000,E1 345.644} C_DIS
LIN {X -0.003,Y -173.298,Z 1729.892,A 0.000,B 0.000,C 90.000,E1 340.496} C_DIS
LIN {X -0.054,Y -176.711,Z 1729.868,A 0.000,B 0.000,C 90.000,E1 336.230} C_DIS
LIN {X -0.033,Y -180.976,Z 1729.844,A 0.000,B 0.000,C 90.000,E1 331.975} C_DIS
LIN {X -0.055,Y -185.290,Z 1729.826,A 0.000,B 0.000,C 90.000,E1 328.614} C_DIS
LIN {X 0.007,Y -190.519,Z 1729.807,A 0.000,B 0.000,C 90.000,E1 325.261} C_DIS
LIN {X 0.089,Y -195.150,Z 1729.793,A 0.000,B 0.000,C 90.000,E1 322.763} C_DIS
LIN {X -0.052,Y -200.517,Z 1729.780,A 0.000,B 0.000,C 90.000,E1 320.356} C_DIS
LIN {X -0.104,Y -207.618,Z 1729.764,A 0.000,B 0.000,C 90.000,E1 317.553} C_DIS
LIN {X -0.010,Y -215.712,Z 1729.749,A 0.000,B 0.000,C 90.000,E1 314.757} C_DIS
LIN {X -0.026,Y -222.223,Z 1729.738,A 0.000,B 0.000,C 90.000,E1 312.813} C_DIS
LIN {X -0.087,Y -229.453,Z 1729.727,A 0.000,B 0.000,C 90.000,E1 310.906} C_DIS
LIN {X 0.004,Y -237.559,Z 1729.717,A 0.000,B 0.000,C 90.000,E1 308.991} C_DIS
LIN {X -0.112,Y -246.618,Z 1729.706,A 0.000,B 0.000,C 90.000,E1 307.156} C_DIS
LIN {X -0.033,Y -256.710,Z 1729.696,A 0.000,B 0.000,C 90.000,E1 305.311} C_DIS
LIN {X -0.048,Y -274.569,Z 1729.680,A 0.000,B 0.000,C 90.000,E1 302.467} C_DIS
LIN {X -0.047,Y -294.011,Z 1729.665,A 0.000,B 0.000,C 90.000,E1 299.716} C_DIS
LIN {X -0.048,Y -309.354,Z 1729.654,A 0.000,B 0.000,C 90.000,E1 297.719} C_DIS
LIN {X -0.027,Y -325.155,Z 1729.643,A 0.000,B 0.000,C 90.000,E1 295.771} C_DIS
LIN {X -0.108,Y -340.947,Z 1729.633,A 0.000,B 0.000,C 90.000,E1 293.898} C_DIS
LIN {X 0.063,Y -351.309,Z 1729.626,A 0.000,B 0.000,C 90.000,E1 292.642} C_DIS
LIN {X -0.077,Y -363.775,Z 1729.617,A 0.000,B 0.000,C 90.000,E1 291.153} C_DIS
LIN {X 0.011,Y -371.013,Z 1729.613,A 0.000,B 0.000,C 90.000,E1 290.248} C_DIS
LIN {X -0.188,Y -377.813,Z 1729.608,A 0.000,B 0.000,C 90.000,E1 289.396} C_DIS
LIN {X 0.039,Y -381.868,Z 1729.604,A 0.000,B 0.000,C 90.000,E1 288.779} C_DIS
LIN {X -0.179,Y -387.120,Z 1729.600,A 0.000,B 0.000,C 90.000,E1 287.946} C_DIS
LIN {X 0.107,Y -390.079,Z 1729.596,A 0.000,B 0.000,C 90.000,E1 287.330} C_DIS
LIN {X -0.038,Y -393.722,Z 1729.592,A 0.000,B 0.000,C 90.000,E1 286.496} C_DIS
LIN {X 0.176,Y -395.627,Z 1729.589,A 0.000,B 0.000,C 90.000,E1 285.898} C_DIS
LIN {X -0.090,Y -397.231,Z 1729.585,A 0.000,B 0.000,C 90.000,E1 285.371} C_DIS
LIN {X 0.144,Y -398.460,Z 1729.582,A 0.000,B 0.000,C 90.000,E1 284.773} C_DIS
LIN {X -0.100,Y -399.353,Z 1729.579,A 0.000,B 0.000,C 90.000,E1 284.245} C_DIS
LIN {X 0.149,Y -399.847,Z 1729.576,A 0.000,B 0.000,C 90.000,E1 283.647} C_DIS
LIN {X -0.081,Y -399.980,Z 1729.573,A 0.000,B 0.000,C 90.000,E1 283.119} C_DIS
LIN {X 0.083,Y -399.735,Z 1729.570,A 0.000,B 0.000,C 90.000,E1 282.535} C_DIS
LIN {X -0.142,Y -399.026,Z 1729.567,A 0.000,B 0.000,C 90.000,E1 282.007} C_DIS
LIN {X 0.022,Y -397.842,Z 1729.563,A 0.000,B 0.000,C 90.000,E1 281.422} C_DIS
LIN {X 0.181,Y -396.153,Z 1729.560,A 0.000,B 0.000,C 90.000,E1 280.838} C_DIS
LIN {X -0.057,Y -393.914,Z 1729.557,A 0.000,B 0.000,C 90.000,E1 280.310} C_DIS
LIN {X 0.075,Y -391.094,Z 1729.554,A 0.000,B 0.000,C 90.000,E1 279.726} C_DIS
LIN {X -0.094,Y -377.875,Z 1729.541,A 0.000,B 0.000,C 90.000,E1 277.466} C_DIS
LIN {X -0.114,Y -374.075,Z 1729.538,A 0.000,B 0.000,C 90.000,E1 276.891} C_DIS
LIN {X -0.153,Y -369.744,Z 1729.535,A 0.000,B 0.000,C 90.000,E1 276.315} C_DIS
LIN {X 0.149,Y -364.750,Z 1729.532,A 0.000,B 0.000,C 90.000,E1 275.682} C_DIS
LIN {X 0.079,Y -358.993,Z 1729.528,A 0.000,B 0.000,C 90.000,E1 275.106} C_DIS
LIN {X -0.054,Y -353.109,Z 1729.525,A 0.000,B 0.000,C 90.000,E1 274.588} C_DIS
LIN {X -0.006,Y -347.013,Z 1729.523,A 0.000,B 0.000,C 90.000,E1 274.073} C_DIS
LIN {X -0.041,Y -340.757,Z 1729.520,A 0.000,B 0.000,C 90.000,E1 273.612} C_DIS
LIN {X 0.143,Y -334.453,Z 1729.518,A 0.000,B 0.000,C 90.000,E1 273.154} C_DIS
LIN {X -0.132,Y -327.894,Z 1729.516,A 0.000,B 0.000,C 90.000,E1 272.808} C_DIS
LIN {X 0.149,Y -321.257,Z 1729.514,A 0.000,B 0.000,C 90.000,E1 272.407} C_DIS
LIN {X -0.029,Y -314.343,Z 1729.512,A 0.000,B 0.000,C 90.000,E1 272.121} C_DIS
LIN {X 0.019,Y -307.189,Z 1729.510,A 0.000,B 0.000,C 90.000,E1 271.835} C_DIS
LIN {X 0.116,Y -296.428,Z 1729.508,A 0.000,B 0.000,C 90.000,E1 271.489} C_DIS
LIN {X 0.072,Y -289.060,Z 1729.507,A 0.000,B 0.000,C 90.000,E1 271.318} C_DIS
LIN {X -0.118,Y -281.178,Z 1729.507,A 0.000,B 0.000,C 90.000,E1 271.203} C_DIS
LIN {X 0.097,Y -263.854,Z 1729.505,A 0.000,B 0.000,C 90.000,E1 270.917} C_DIS
LIN {X 0.023,Y -249.256,Z 1729.505,A 0.000,B 0.000,C 90.000,E1 270.802} C_DIS
LIN {X 0.115,Y -241.454,Z 1729.504,A 0.000,B 0.000,C 90.000,E1 270.745} C_DIS
LIN {X 0.054,Y -181.511,Z 1729.504,A 0.000,B 0.000,C 90.000,E1 270.745} C_DIS
LIN {X -0.087,Y -181.533,Z 1729.499,A 0.000,B 0.000,C 90.000,E1 269.885} C_DIS
LIN {X 0.078,Y -180.806,Z 1729.471,A 0.000,B 0.000,C 90.000,E1 264.780} C_DIS
LIN {X -0.025,Y -178.908,Z 1729.443,A 0.000,B 0.000,C 90.000,E1 259.746} C_DIS
LIN {X 0.055,Y -175.951,Z 1729.415,A 0.000,B 0.000,C 90.000,E1 254.629} C_DIS
LIN {X 0.002,Y -175.417,Z 1729.410,A 0.000,B 0.000,C 90.000,E1 253.795} C_DIS
LIN {X 0.005,Y -172.179,Z 1729.386,A 0.000,B 0.000,C 90.000,E1 249.518} C_DIS
LIN {X 0.044,Y -171.650,Z 1729.381,A 0.000,B 0.000,C 90.000,E1 248.646} C_DIS
LIN {X 0.038,Y -167.874,Z 1729.357,A 0.000,B 0.000,C 90.000,E1 244.332} C_DIS
LIN {X -0.018,Y -166.609,Z 1729.348,A 0.000,B 0.000,C 90.000,E1 242.615} C_DIS
LIN {X -0.024,Y -162.597,Z 1729.324,A 0.000,B 0.000,C 90.000,E1 238.250} C_DIS
LIN {X -0.050,Y -161.282,Z 1729.314,A 0.000,B 0.000,C 90.000,E1 236.501} C_DIS
LIN {X -0.015,Y -157.281,Z 1729.289,A 0.000,B 0.000,C 90.000,E1 232.065} C_DIS
LIN {X 0.008,Y -156.000,Z 1729.279,A 0.000,B 0.000,C 90.000,E1 230.275} C_DIS
LIN {X -0.032,Y -152.258,Z 1729.254,A 0.000,B 0.000,C 90.000,E1 225.810} C_DIS
LIN {X -0.010,Y -150.496,Z 1729.239,A 0.000,B 0.000,C 90.000,E1 223.095} C_DIS
LIN {X 0.020,Y -147.221,Z 1729.214,A 0.000,B 0.000,C 90.000,E1 218.543} C_DIS
LIN {X -0.010,Y -145.242,Z 1729.194,A 0.000,B 0.000,C 90.000,E1 214.898} C_DIS
LIN {X 0.031,Y -142.362,Z 1729.163,A 0.000,B 0.000,C 90.000,E1 209.361} C_DIS
LIN {X 0.028,Y -141.748,Z 1729.153,A 0.000,B 0.000,C 90.000,E1 207.513} C_DIS
LIN {X -0.047,Y -139.492,Z 1729.117,A 0.000,B 0.000,C 90.000,E1 201.046} C_DIS
LIN {X -0.010,Y -138.996,Z 1729.101,A 0.000,B 0.000,C 90.000,E1 198.236} C_DIS
LIN {X -0.053,Y -138.337,Z 1729.055,A 0.000,B 0.000,C 90.000,E1 189.849} C_DIS
LIN {X -0.031,Y -139.414,Z 1729.008,A 0.000,B 0.000,C 90.000,E1 181.432} C_DIS
LIN {X 0.023,Y -141.328,Z 1728.972,A 0.000,B 0.000,C 90.000,E1 174.894} C_DIS
LIN {X -0.021,Y -142.686,Z 1728.956,A 0.000,B 0.000,C 90.000,E1 172.129} C_DIS
LIN {X -0.041,Y -145.046,Z 1728.931,A 0.000,B 0.000,C 90.000,E1 167.521} C_DIS
LIN {X -0.044,Y -147.672,Z 1728.910,A 0.000,B 0.000,C 90.000,E1 163.850} C_DIS
LIN {X -0.009,Y -150.314,Z 1728.890,A 0.000,B 0.000,C 90.000,E1 160.188} C_DIS
LIN {X 0.063,Y -153.727,Z 1728.870,A 0.000,B 0.000,C 90.000,E1 156.538} C_DIS
LIN {X -0.085,Y -157.141,Z 1728.850,A 0.000,B 0.000,C 90.000,E1 152.999} C_DIS
LIN {X -0.010,Y -161.289,Z 1728.830,A 0.000,B 0.000,C 90.000,E1 149.410} C_DIS
LIN {X 0.007,Y -164.405,Z 1728.815,A 0.000,B 0.000,C 90.000,E1 146.755} C_DIS
LIN {X 0.004,Y -169.086,Z 1728.796,A 0.000,B 0.000,C 90.000,E1 143.256} C_DIS
LIN {X -0.045,Y -171.643,Z 1728.786,A 0.000,B 0.000,C 90.000,E1 141.537} C_DIS
LIN {X 0.001,Y -176.604,Z 1728.767,A 0.000,B 0.000,C 90.000,E1 138.081} C_DIS
LIN {X 0.003,Y -180.903,Z 1728.753,A 0.000,B 0.000,C 90.000,E1 135.526} C_DIS
LIN {X -0.006,Y -186.319,Z 1728.734,A 0.000,B 0.000,C 90.000,E1 132.162} C_DIS
LIN {X 0.061,Y -190.953,Z 1728.720,A 0.000,B 0.000,C 90.000,E1 129.644} C_DIS
LIN {X -0.019,Y -196.724,Z 1728.702,A 0.000,B 0.000,C 90.000,E1 126.377} C_DIS
LIN {X 0.011,Y -199.971,Z 1728.693,A 0.000,B 0.000,C 90.000,E1 124.739} C_DIS
LIN {X -0.005,Y -207.474,Z 1728.671,A 0.000,B 0.000,C 90.000,E1 120.718} C_DIS
LIN {X -0.026,Y -209.845,Z 1728.664,A 0.000,B 0.000,C 90.000,E1 119.589} C_DIS
LIN {X 0.184,Y -334.351,Z 1728.664,A 0.000,B 0.000,C 90.000,E1 119.539} C_DIS
LIN {X -0.012,Y -336.419,Z 1728.664,A 0.000,B 0.000,C 90.000,E1 119.539} C_DIS
LIN {X -0.011,Y -340.956,Z 1728.663,A 0.000,B 0.000,C 90.000,E1 119.333} C_DIS
LIN {X -0.011,Y -343.509,Z 1728.662,A 0.000,B 0.000,C 90.000,E1 119.127} C_DIS
LIN {X -0.196,Y -347.290,Z 1728.659,A 0.000,B 0.000,C 90.000,E1 118.693} C_DIS
LIN {X -0.031,Y -349.020,Z 1728.657,A 0.000,B 0.000,C 90.000,E1 118.359} C_DIS
LIN {X -0.009,Y -363.487,Z 1728.641,A 0.000,B 0.000,C 90.000,E1 115.335} C_DIS
LIN {X -0.105,Y -378.092,Z 1728.626,A 0.000,B 0.000,C 90.000,E1 112.695} C_DIS
LIN {X -0.022,Y -392.462,Z 1728.613,A 0.000,B 0.000,C 90.000,E1 110.375} C_DIS
LIN {X -0.072,Y -408.243,Z 1728.601,A 0.000,B 0.000,C 90.000,E1 108.127} C_DIS
LIN {X 0.136,Y -425.543,Z 1728.588,A 0.000,B 0.000,C 90.000,E1 105.898} C_DIS
LIN {X 0.007,Y -444.483,Z 1728.577,A 0.000,B 0.000,C 90.000,E1 103.772} C_DIS
LIN {X -0.098,Y -464.459,Z 1728.565,A 0.000,B 0.000,C 90.000,E1 101.771} C_DIS
LIN {X 0.147,Y -487.567,Z 1728.554,A 0.000,B 0.000,C 90.000,E1 99.670} C_DIS
LIN {X 0.058,Y -508.500,Z 1728.544,A 0.000,B 0.000,C 90.000,E1 97.992} C_DIS
LIN {X -0.158,Y -510.447,Z 1728.543,A 0.000,B 0.000,C 90.000,E1 97.814} C_DIS
LIN {X 0.230,Y -512.198,Z 1728.542,A 0.000,B 0.000,C 90.000,E1 97.530} C_DIS
LIN {X 0.179,Y -513.508,Z 1728.541,A 0.000,B 0.000,C 90.000,E1 97.296} C_DIS
LIN {X 0.031,Y -515.112,Z 1728.538,A 0.000,B 0.000,C 90.000,E1 96.834} C_DIS
LIN {X -0.111,Y -515.615,Z 1728.535,A 0.000,B 0.000,C 90.000,E1 96.372} C_DIS
LIN {X 0.268,Y -515.099,Z 1728.533,A 0.000,B 0.000,C 90.000,E1 95.853} C_DIS
LIN {X 0.134,Y -513.476,Z 1728.530,A 0.000,B 0.000,C 90.000,E1 95.391} C_DIS
LIN {X 0.044,Y -512.155,Z 1728.529,A 0.000,B 0.000,C 90.000,E1 95.163} C_DIS
LIN {X -0.087,Y -499.573,Z 1728.519,A 0.000,B 0.000,C 90.000,E1 93.498} C_DIS
LIN {X 0.155,Y -488.766,Z 1728.511,A 0.000,B 0.000,C 90.000,E1 92.007} C_DIS
LIN {X -0.138,Y -474.139,Z 1728.500,A 0.000,B 0.000,C 90.000,E1 90.057} C_DIS
LIN {X -0.082,Y -461.321,Z 1728.490,A 0.000,B 0.000,C 90.000,E1 88.282} C_DIS
LIN {X 0.203,Y -448.460,Z 1728.480,A 0.000,B 0.000,C 90.000,E1 86.445} C_DIS
LIN {X -0.217,Y -435.614,Z 1728.470,A 0.000,B 0.000,C 90.000,E1 84.666} C_DIS
LIN {X 0.216,Y -421.003,Z 1728.458,A 0.000,B 0.000,C 90.000,E1 82.470} C_DIS
LIN {X 0.212,Y -401.716,Z 1728.442,A 0.000,B 0.000,C 90.000,E1 79.454} C_DIS
LIN {X 0.153,Y -385.307,Z 1728.426,A 0.000,B 0.000,C 90.000,E1 76.645} C_DIS
LIN {X 0.158,Y -372.689,Z 1728.413,A 0.000,B 0.000,C 90.000,E1 74.338} C_DIS
LIN {X 0.067,Y -360.348,Z 1728.400,A 0.000,B 0.000,C 90.000,E1 72.000} C_DIS
LIN {X -0.120,Y -344.106,Z 1728.382,A 0.000,B 0.000,C 90.000,E1 68.720} C_DIS
LIN {X 0.054,Y -334.163,Z 1728.370,A 0.000,B 0.000,C 90.000,E1 66.538} C_DIS
LIN {X 0.047,Y -321.508,Z 1728.354,A 0.000,B 0.000,C 90.000,E1 63.717} C_DIS
LIN {X -0.056,Y -313.332,Z 1728.343,A 0.000,B 0.000,C 90.000,E1 61.820} C_DIS
LIN {X 0.013,Y -303.692,Z 1728.331,A 0.000,B 0.000,C 90.000,E1 59.537} C_DIS
LIN {X -0.089,Y -294.040,Z 1728.318,A 0.000,B 0.000,C 90.000,E1 57.248} C_DIS
LIN {X -0.052,Y -285.709,Z 1728.307,A 0.000,B 0.000,C 90.000,E1 55.229} C_DIS
LIN {X -0.055,Y -275.919,Z 1728.293,A 0.000,B 0.000,C 90.000,E1 52.844} C_DIS
LIN {X -0.166,Y -266.148,Z 1728.280,A 0.000,B 0.000,C 90.000,E1 50.436} C_DIS
LIN {X 0.060,Y -255.154,Z 1728.264,A 0.000,B 0.000,C 90.000,E1 47.553} C_DIS
LIN {X 0.145,Y -243.219,Z 1728.246,A 0.000,B 0.000,C 90.000,E1 44.271} C_DIS
LIN {X -0.086,Y -231.946,Z 1728.228,A 0.000,B 0.000,C 90.000,E1 40.987} C_DIS
LIN {X -0.010,Y -222.671,Z 1728.211,A 0.000,B 0.000,C 90.000,E1 37.935} C_DIS
LIN {X 0.016,Y -215.284,Z 1728.196,A 0.000,B 0.000,C 90.000,E1 35.231} C_DIS
LIN {X 0.073,Y -207.636,Z 1728.178,A 0.000,B 0.000,C 90.000,E1 32.084} C_DIS
LIN {X -0.096,Y -200.634,Z 1728.161,A 0.000,B 0.000,C 90.000,E1 28.949} C_DIS
LIN {X -0.099,Y -194.370,Z 1728.143,A 0.000,B 0.000,C 90.000,E1 25.720} C_DIS
END
